LIN {X 0,Y 418.251,Z 298.382,A -85,B 0,C 180,E1 -10100.663,E2 -10100.663} C_VEL
LIN {X 0,Y 418.279,Z 298.377,A -85,B 0,C 180,E1 -10103.782,E2 -10103.782} C_VEL
LIN {X 0,Y 418.312,Z 298.374,A -85,B 0,C 180,E1 -10107.07,E2 -10107.07} C_VEL
LIN {X 0,Y 418.246,Z 298.384,A -85,B 0,C 180,E1 -10110.272,E2 -10110.272} C_VEL
LIN {X 0,Y 418.249,Z 298.383,A -85,B 0,C 180,E1 -10113.677,E2 -10113.677} C_VEL
LIN {X 0,Y 418.241,Z 298.386,A -85,B 0,C 180,E1 -10117.224,E2 -10117.224} C_VEL
LIN {X 0,Y 418.248,Z 298.385,A -85,B 0,C 180,E1 -10119.682,E2 -10119.682} C_VEL
LIN {X 0,Y 418.231,Z 298.386,A -85,B 0,C 180,E1 -10122.321,E2 -10122.321} C_VEL
LIN {X 0,Y 418.237,Z 298.39,A -85,B 0,C 180,E1 -10125.109,E2 -10125.109} C_VEL
LIN {X 0,Y 418.242,Z 298.386,A -85,B 0,C 180,E1 -10127.767,E2 -10127.767} C_VEL
LIN {X 0,Y 418.247,Z 298.385,A -85,B 0,C 180,E1 -10130.62,E2 -10130.62} C_VEL
LIN {X 0,Y 418.245,Z 298.393,A -85,B 0,C 180,E1 -10133.976,E2 -10133.976} C_VEL
LIN {X 0,Y 418.26,Z 298.389,A -85,B 0,C 180,E1 -10137.156,E2 -10137.156} C_VEL
LIN {X 0,Y 418.271,Z 298.384,A -85,B 0,C 180,E1 -10140.895,E2 -10140.895} C_VEL
LIN {X 0,Y 418.335,Z 298.472,A -85,B 0,C 180,E1 -10142.493,E2 -10142.493} C_VEL
LIN {X 0,Y 420.755,Z 310.164,A -85,B 0,C 180,E1 -10144.936,E2 -10144.936} C_VEL
LIN {X 0,Y 421.189,Z 314.876,A -85,B 0,C 180,E1 -10145.87,E2 -10145.87} C_VEL
LIN {X 0,Y 420.116,Z 333.869,A -85,B 0,C 180,E1 -10149.433,E2 -10149.433} C_VEL
LIN {X 0,Y 419.738,Z 340.825,A -85,B 0,C 180,E1 -10150.723,E2 -10150.723} C_VEL
LIN {X 0,Y 423.765,Z 366.097,A -85,B 0,C 180,E1 -10151.423,E2 -10151.423} C_VEL
LIN {X 0,Y 423.972,Z 371.55,A -85,B 0,C 180,E1 -10151.538,E2 -10151.538} C_VEL
LIN {X 0,Y 422.818,Z 450.347,A -85,B 0,C 180,E1 -10152.995,E2 -10152.995} C_VEL
LIN {X 0,Y 422.307,Z 463.22,A -85,B 0,C 180,E1 -10153.41,E2 -10153.41} C_VEL
LIN {X 0,Y 421.668,Z 475.247,A -85,B 0,C 180,E1 -10153.975,E2 -10153.975} C_VEL
LIN {X 0,Y 420.931,Z 487.489,A -85,B 0,C 180,E1 -10154.753,E2 -10154.753} C_VEL
LIN {X 0,Y 420.211,Z 498.894,A -85,B 0,C 180,E1 -10155.697,E2 -10155.697} C_VEL
LIN {X 0,Y 419.4,Z 509.61,A -85,B 0,C 180,E1 -10156.801,E2 -10156.801} C_VEL
LIN {X 0,Y 418.827,Z 518.21,A -85,B 0,C 180,E1 -10157.892,E2 -10157.892} C_VEL
LIN {X 0,Y 418.085,Z 527.537,A -85,B 0,C 180,E1 -10159.344,E2 -10159.344} C_VEL
LIN {X 0,Y 417.632,Z 535.048,A -85,B 0,C 180,E1 -10160.8,E2 -10160.8} C_VEL
LIN {X 0,Y 417.351,Z 541.088,A -85,B 0,C 180,E1 -10162.257,E2 -10162.257} C_VEL
LIN {X 0,Y 417.165,Z 545.849,A -85,B 0,C 180,E1 -10163.708,E2 -10163.708} C_VEL
LIN {X 0,Y 417.107,Z 549.513,A -85,B 0,C 180,E1 -10165.167,E2 -10165.167} C_VEL
LIN {X 0,Y 417.016,Z 551.381,A -85,B 0,C 180,E1 -10166.134,E2 -10166.134} C_VEL
LIN {X 0,Y 417.031,Z 552.79,A -85,B 0,C 180,E1 -10167.101,E2 -10167.101} C_VEL
LIN {X 0,Y 417.069,Z 553.797,A -85,B 0,C 180,E1 -10168.068,E2 -10168.068} C_VEL
LIN {X 0,Y 417.032,Z 554.406,A -85,B 0,C 180,E1 -10169.034,E2 -10169.034} C_VEL
LIN {X 0,Y 417.028,Z 554.587,A -85,B 0,C 180,E1 -10169.999,E2 -10169.999} C_VEL
LIN {X 0,Y 417.032,Z 554.344,A -85,B 0,C 180,E1 -10170.965,E2 -10170.965} C_VEL
LIN {X 0,Y 417.069,Z 553.708,A -85,B 0,C 180,E1 -10171.931,E2 -10171.931} C_VEL
LIN {X 0,Y 417.033,Z 552.671,A -85,B 0,C 180,E1 -10172.897,E2 -10172.897} C_VEL
LIN {X 0,Y 417.016,Z 551.183,A -85,B 0,C 180,E1 -10173.865,E2 -10173.865} C_VEL
LIN {X 0,Y 417.118,Z 548.137,A -85,B 0,C 180,E1 -10175.317,E2 -10175.317} C_VEL
LIN {X 0,Y 417.23,Z 544.008,A -85,B 0,C 180,E1 -10176.771,E2 -10176.771} C_VEL
LIN {X 0,Y 417.491,Z 537.664,A -85,B 0,C 180,E1 -10178.47,E2 -10178.47} C_VEL
LIN {X 0,Y 417.859,Z 530.747,A -85,B 0,C 180,E1 -10179.926,E2 -10179.926} C_VEL
LIN {X 0,Y 418.282,Z 523.68,A -85,B 0,C 180,E1 -10181.14,E2 -10181.14} C_VEL
LIN {X 0,Y 418.918,Z 515.169,A -85,B 0,C 180,E1 -10182.35,E2 -10182.35} C_VEL
LIN {X 0,Y 419.594,Z 504.638,A -85,B 0,C 180,E1 -10183.561,E2 -10183.561} C_VEL
LIN {X 0,Y 420.256,Z 492.783,A -85,B 0,C 180,E1 -10184.651,E2 -10184.651} C_VEL
LIN {X 0,Y 420.974,Z 480.89,A -85,B 0,C 180,E1 -10185.492,E2 -10185.492} C_VEL
LIN {X 0,Y 421.638,Z 468.569,A -85,B 0,C 180,E1 -10186.149,E2 -10186.149} C_VEL
LIN {X 0,Y 422.184,Z 456.025,A -85,B 0,C 180,E1 -10186.625,E2 -10186.625} C_VEL
LIN {X 0,Y 422.534,Z 441.559,A -85,B 0,C 180,E1 -10186.953,E2 -10186.953} C_VEL
LIN {X 0,Y 423.317,Z 366.905,A -85,B 0,C 180,E1 -10188.298,E2 -10188.298} C_VEL
LIN {X 0,Y 419.561,Z 342.148,A -85,B 0,C 180,E1 -10188.937,E2 -10188.937} C_VEL
LIN {X 0,Y 420.631,Z 325.944,A -85,B 0,C 180,E1 -10192.081,E2 -10192.081} C_VEL
LIN {X 0,Y 421.354,Z 314.259,A -85,B 0,C 180,E1 -10194.381,E2 -10194.381} C_VEL
LIN {X 0,Y 419.417,Z 303.717,A -85,B 0,C 180,E1 -10196.63,E2 -10196.63} C_VEL
LIN {X 0,Y 418.333,Z 298.377,A -85,B 0,C 180,E1 -10197.821,E2 -10197.821} C_VEL
LIN {X 0,Y 418.209,Z 298.387,A -85,B 0,C 180,E1 -10201.395,E2 -10201.395} C_VEL
LIN {X 0,Y 418.263,Z 298.383,A -85,B 0,C 180,E1 -10204.58,E2 -10204.58} C_VEL
LIN {X 0,Y 418.223,Z 298.387,A -85,B 0,C 180,E1 -10207.832,E2 -10207.832} C_VEL
LIN {X 0,Y 418.219,Z 298.387,A -85,B 0,C 180,E1 -10210.947,E2 -10210.947} C_VEL
LIN {X 0,Y 418.206,Z 298.387,A -85,B 0,C 180,E1 -10213.729,E2 -10213.729} C_VEL
LIN {X 0,Y 418.212,Z 298.393,A -85,B 0,C 180,E1 -10216.449,E2 -10216.449} C_VEL
LIN {X 0,Y 418.221,Z 298.387,A -85,B 0,C 180,E1 -10219.129,E2 -10219.129} C_VEL
LIN {X 0,Y 418.231,Z 298.385,A -85,B 0,C 180,E1 -10222.165,E2 -10222.165} C_VEL
LIN {X 0,Y 418.261,Z 298.381,A -85,B 0,C 180,E1 -10225.419,E2 -10225.419} C_VEL
LIN {X 0,Y 418.207,Z 298.391,A -85,B 0,C 180,E1 -10228.604,E2 -10228.604} C_VEL
LIN {X 0,Y 418.286,Z 298.377,A -85,B 0,C 180,E1 -10231.936,E2 -10231.936} C_VEL
LIN {X 0,Y 418.284,Z 298.383,A -85,B 0,C 180,E1 -10235.162,E2 -10235.162} C_VEL
LIN {X 0,Y 418.228,Z 298.384,A -85,B 0,C 180,E1 -10238.303,E2 -10238.303} C_VEL
LIN {X 0,Y 418.278,Z 298.383,A -85,B 0,C 180,E1 -10241.383,E2 -10241.383} C_VEL
LIN {X 0,Y 418.297,Z 298.375,A -85,B 0,C 180,E1 -10244.406,E2 -10244.406} C_VEL
LIN {X 0,Y 418.35,Z 298.377,A -85,B 0,C 180,E1 -10247.386,E2 -10247.386} C_VEL
LIN {X 0,Y 418.335,Z 298.371,A -85,B 0,C 180,E1 -10250.329,E2 -10250.329} C_VEL
LIN {X 0,Y 418.507,Z 298.35,A -85,B 0,C 180,E1 -10252.279,E2 -10252.279} C_VEL
LIN {X 0,Y 418.507,Z 298.35,A -85,B 0,C 180,E1 -10254.217,E2 -10254.217} C_VEL
LIN {X 0,Y 418.536,Z 298.348,A -85,B 0,C 180,E1 -10258.076,E2 -10258.076} C_VEL
LIN {X 0,Y 418.664,Z 298.334,A -85,B 0,C 180,E1 -10260,E2 -10260} C_VEL
LIN {X 0,Y 418.496,Z 298.35,A -85,B 0,C 180,E1 -10262.888,E2 -10262.888} C_VEL
LIN {X 0,Y 418.452,Z 298.356,A -85,B 0,C 180,E1 -10266.52,E2 -10266.52} C_VEL
LIN {X 0,Y 418.335,Z 298.374,A -85,B 0,C 180,E1 -10269.672,E2 -10269.672} C_VEL
LIN {X 0,Y 418.341,Z 298.37,A -85,B 0,C 180,E1 -10273.001,E2 -10273.001} C_VEL
LIN {X 0,Y 418.307,Z 298.376,A -85,B 0,C 180,E1 -10276.736,E2 -10276.736} C_VEL
LIN {X 0,Y 418.265,Z 298.382,A -85,B 0,C 180,E1 -10279.791,E2 -10279.791} C_VEL
LIN {X 0,Y 418.227,Z 298.387,A -85,B 0,C 180,E1 -10282.737,E2 -10282.737} C_VEL
LIN {X 0,Y 418.233,Z 298.385,A -85,B 0,C 180,E1 -10285.907,E2 -10285.907} C_VEL
LIN {X 0,Y 418.257,Z 298.381,A -85,B 0,C 180,E1 -10289.163,E2 -10289.163} C_VEL
LIN {X 0,Y 418.254,Z 298.386,A -85,B 0,C 180,E1 -10292.845,E2 -10292.845} C_VEL
LIN {X 0,Y 418.242,Z 298.384,A -85,B 0,C 180,E1 -10296.239,E2 -10296.239} C_VEL
LIN {X 0,Y 418.231,Z 298.384,A -85,B 0,C 180,E1 -10299.685,E2 -10299.685} C_VEL
LIN {X 0,Y 418.221,Z 298.386,A -85,B 0,C 180,E1 -10302.321,E2 -10302.321} C_VEL
LIN {X 0,Y 418.234,Z 298.389,A -85,B 0,C 180,E1 -10305.11,E2 -10305.11} C_VEL
LIN {X 0,Y 418.221,Z 298.385,A -85,B 0,C 180,E1 -10307.766,E2 -10307.766} C_VEL
LIN {X 0,Y 418.239,Z 298.385,A -85,B 0,C 180,E1 -10311.558,E2 -10311.558} C_VEL
LIN {X 0,Y 418.258,Z 298.387,A -85,B 0,C 180,E1 -10315.16,E2 -10315.16} C_VEL
LIN {X 0,Y 418.245,Z 298.387,A -85,B 0,C 180,E1 -10317.473,E2 -10317.473} C_VEL
LIN {X 0,Y 418.262,Z 298.382,A -85,B 0,C 180,E1 -10320.898,E2 -10320.898} C_VEL
LIN {X 0,Y 418.225,Z 298.385,A -85,B 0,C 180,E1 -10324.094,E2 -10324.094} C_VEL
LIN {X 0,Y 418.229,Z 298.388,A -85,B 0,C 180,E1 -10327.264,E2 -10327.264} C_VEL
LIN {X 0,Y 418.285,Z 298.377,A -85,B 0,C 180,E1 -10330.365,E2 -10330.365} C_VEL
LIN {X 0,Y 418.318,Z 298.377,A -85,B 0,C 180,E1 -10333.405,E2 -10333.405} C_VEL
LIN {X 0,Y 418.349,Z 298.369,A -85,B 0,C 180,E1 -10337.001,E2 -10337.001} C_VEL
LIN {X 0,Y 418.323,Z 298.375,A -85,B 0,C 180,E1 -10340.329,E2 -10340.329} C_VEL
LIN {X 0,Y 418.445,Z 298.357,A -85,B 0,C 180,E1 -10343.249,E2 -10343.249} C_VEL
LIN {X 0,Y 418.315,Z 298.373,A -85,B 0,C 180,E1 -10345.182,E2 -10345.182} C_VEL
LIN {X 0,Y 418.533,Z 298.354,A -85,B 0,C 180,E1 -10348.076,E2 -10348.076} C_VEL
LIN {X 0,Y 418.41,Z 298.362,A -85,B 0,C 180,E1 -10350.963,E2 -10350.963} C_VEL
LIN {X 0,Y 418.457,Z 298.356,A -85,B 0,C 180,E1 -10352.889,E2 -10352.889} C_VEL
LIN {X 0,Y 418.473,Z 298.355,A -85,B 0,C 180,E1 -10355.784,E2 -10355.784} C_VEL
LIN {X 0,Y 418.369,Z 298.371,A -85,B 0,C 180,E1 -10358.696,E2 -10358.696} C_VEL
LIN {X 0,Y 418.349,Z 298.376,A -85,B 0,C 180,E1 -10362.615,E2 -10362.615} C_VEL
LIN {X 0,Y 418.305,Z 298.375,A -85,B 0,C 180,E1 -10363.316,E2 -10363.316} C_VEL
LIN {X 0,Y 417.583,Z 298.469,A -85,B 0,C 180,E1 -10364.12,E2 -10364.12} C_VEL
LIN {X 0,Y 414.695,Z 298.824,A -85,B 0,C 180,E1 -10365.425,E2 -10365.425} C_VEL
LIN {X 0,Y 412.29,Z 299.13,A -85,B 0,C 180,E1 -10366.479,E2 -10366.479} C_VEL
LIN {X 0,Y 411.271,Z 299.252,A -85,B 0,C 180,E1 -10367.293,E2 -10367.293} C_VEL
LIN {X 0,Y 411.194,Z 299.26,A -85,B 0,C 180,E1 -10367.569,E2 -10367.569} C_VEL
LIN {X 0,Y 411.192,Z 299.266,A -85,B 0,C 180,E1 -10371.035,E2 -10371.035} C_VEL
LIN {X 0,Y 411.257,Z 299.456,A -85,B 0,C 180,E1 -10374.586,E2 -10374.586} C_VEL
LIN {X 0,Y 413.05,Z 309.513,A -85,B 0,C 180,E1 -10377.075,E2 -10377.075} C_VEL
LIN {X 0,Y 412.957,Z 312.92,A -85,B 0,C 180,E1 -10377.868,E2 -10377.868} C_VEL
LIN {X 0,Y 416.883,Z 333.61,A -85,B 0,C 180,E1 -10378.441,E2 -10378.441} C_VEL
LIN {X 0,Y 415.656,Z 420.17,A -85,B 0,C 180,E1 -10380.043,E2 -10380.043} C_VEL
LIN {X 0,Y 415.177,Z 433.503,A -85,B 0,C 180,E1 -10380.479,E2 -10380.479} C_VEL
LIN {X 0,Y 414.747,Z 446.548,A -85,B 0,C 180,E1 -10381.12,E2 -10381.12} C_VEL
LIN {X 0,Y 414.027,Z 458.605,A -85,B 0,C 180,E1 -10381.924,E2 -10381.924} C_VEL
LIN {X 0,Y 413.292,Z 470.672,A -85,B 0,C 180,E1 -10382.968,E2 -10382.968} C_VEL
LIN {X 0,Y 412.789,Z 480.02,A -85,B 0,C 180,E1 -10383.981,E2 -10383.981} C_VEL
LIN {X 0,Y 412.08,Z 489.365,A -85,B 0,C 180,E1 -10385.218,E2 -10385.218} C_VEL
LIN {X 0,Y 411.368,Z 498.536,A -85,B 0,C 180,E1 -10386.724,E2 -10386.724} C_VEL
LIN {X 0,Y 410.855,Z 506.345,A -85,B 0,C 180,E1 -10388.349,E2 -10388.349} C_VEL
LIN {X 0,Y 410.478,Z 512.736,A -85,B 0,C 180,E1 -10390.066,E2 -10390.066} C_VEL
LIN {X 0,Y 410.236,Z 516.777,A -85,B 0,C 180,E1 -10391.476,E2 -10391.476} C_VEL
LIN {X 0,Y 410.003,Z 520.577,A -85,B 0,C 180,E1 -10393.287,E2 -10393.287} C_VEL
LIN {X 0,Y 409.832,Z 523.05,A -85,B 0,C 180,E1 -10395.324,E2 -10395.324} C_VEL
LIN {X 0,Y 409.822,Z 523.739,A -85,B 0,C 180,E1 -10396.688,E2 -10396.688} C_VEL
LIN {X 0,Y 409.804,Z 523.686,A -85,B 0,C 180,E1 -10398.022,E2 -10398.022} C_VEL
LIN {X 0,Y 409.849,Z 522.874,A -85,B 0,C 180,E1 -10399.336,E2 -10399.336} C_VEL
LIN {X 0,Y 410.076,Z 520.348,A -85,B 0,C 180,E1 -10401.277,E2 -10401.277} C_VEL
LIN {X 0,Y 410.365,Z 516.265,A -85,B 0,C 180,E1 -10403.171,E2 -10403.171} C_VEL
LIN {X 0,Y 410.748,Z 511.185,A -85,B 0,C 180,E1 -10404.845,E2 -10404.845} C_VEL
LIN {X 0,Y 411.254,Z 504.312,A -85,B 0,C 180,E1 -10406.556,E2 -10406.556} C_VEL
LIN {X 0,Y 411.871,Z 496.64,A -85,B 0,C 180,E1 -10408.064,E2 -10408.064} C_VEL
LIN {X 0,Y 412.497,Z 489.141,A -85,B 0,C 180,E1 -10409.26,E2 -10409.26} C_VEL
LIN {X 0,Y 413.144,Z 480.198,A -85,B 0,C 180,E1 -10410.441,E2 -10410.441} C_VEL
LIN {X 0,Y 413.989,Z 469.091,A -85,B 0,C 180,E1 -10411.618,E2 -10411.618} C_VEL
LIN {X 0,Y 414.697,Z 458.601,A -85,B 0,C 180,E1 -10412.51,E2 -10412.51} C_VEL
LIN {X 0,Y 415.357,Z 447.305,A -85,B 0,C 180,E1 -10413.267,E2 -10413.267} C_VEL
LIN {X 0,Y 415.837,Z 434.749,A -85,B 0,C 180,E1 -10413.896,E2 -10413.896} C_VEL
LIN {X 0,Y 416.258,Z 422.566,A -85,B 0,C 180,E1 -10414.314,E2 -10414.314} C_VEL
LIN {X 0,Y 416.73,Z 393.125,A -85,B 0,C 180,E1 -10414.896,E2 -10414.896} C_VEL
LIN {X 0,Y 417.771,Z 332.851,A -85,B 0,C 180,E1 -10416.022,E2 -10416.022} C_VEL
LIN {X 0,Y 413.467,Z 312.572,A -85,B 0,C 180,E1 -10416.669,E2 -10416.669} C_VEL
LIN {X 0,Y 413.236,Z 308.374,A -85,B 0,C 180,E1 -10417.501,E2 -10417.501} C_VEL
LIN {X 0,Y 411.241,Z 299.26,A -85,B 0,C 180,E1 -10419.426,E2 -10419.426} C_VEL
LIN {X 0,Y 411.266,Z 299.262,A -85,B 0,C 180,E1 -10423.131,E2 -10423.131} C_VEL
LIN {X 0,Y 411.308,Z 299.252,A -85,B 0,C 180,E1 -10426.896,E2 -10426.896} C_VEL
LIN {X 0,Y 411.294,Z 299.253,A -85,B 0,C 180,E1 -10430.161,E2 -10430.161} C_VEL
LIN {X 0,Y 411.485,Z 299.23,A -85,B 0,C 180,E1 -10432.146,E2 -10432.146} C_VEL
LIN {X 0,Y 411.473,Z 299.232,A -85,B 0,C 180,E1 -10434.118,E2 -10434.118} C_VEL
LIN {X 0,Y 411.513,Z 299.224,A -85,B 0,C 180,E1 -10438.042,E2 -10438.042} C_VEL
LIN {X 0,Y 411.642,Z 299.21,A -85,B 0,C 180,E1 -10440,E2 -10440} C_VEL
LIN {X 0,Y 411.459,Z 299.229,A -85,B 0,C 180,E1 -10442.937,E2 -10442.937} C_VEL
LIN {X 0,Y 411.46,Z 299.234,A -85,B 0,C 180,E1 -10445.882,E2 -10445.882} C_VEL
LIN {X 0,Y 411.353,Z 299.242,A -85,B 0,C 180,E1 -10448.845,E2 -10448.845} C_VEL
LIN {X 0,Y 411.285,Z 299.252,A -85,B 0,C 180,E1 -10451.833,E2 -10451.833} C_VEL
LIN {X 0,Y 411.263,Z 299.256,A -85,B 0,C 180,E1 -10454.852,E2 -10454.852} C_VEL
LIN {X 0,Y 411.247,Z 299.252,A -85,B 0,C 180,E1 -10457.915,E2 -10457.915} C_VEL
LIN {X 0,Y 411.198,Z 299.26,A -85,B 0,C 180,E1 -10461.034,E2 -10461.034} C_VEL
LIN {X 0,Y 411.222,Z 299.258,A -85,B 0,C 180,E1 -10464.216,E2 -10464.216} C_VEL
LIN {X 0,Y 411.261,Z 299.249,A -85,B 0,C 180,E1 -10467.477,E2 -10467.477} C_VEL
LIN {X 0,Y 411.191,Z 299.264,A -85,B 0,C 180,E1 -10470.847,E2 -10470.847} C_VEL
LIN {X 0,Y 411.206,Z 299.26,A -85,B 0,C 180,E1 -10474.333,E2 -10474.333} C_VEL
LIN {X 0,Y 411.195,Z 299.26,A -85,B 0,C 180,E1 -10477.974,E2 -10477.974} C_VEL
LIN {X 0,Y 411.165,Z 299.268,A -85,B 0,C 180,E1 -10481.228,E2 -10481.228} C_VEL
LIN {X 0,Y 411.178,Z 299.265,A -85,B 0,C 180,E1 -10484.49,E2 -10484.49} C_VEL
LIN {X 0,Y 411.179,Z 299.264,A -85,B 0,C 180,E1 -10488.194,E2 -10488.194} C_VEL
LIN {X 0,Y 411.213,Z 299.261,A -85,B 0,C 180,E1 -10490.775,E2 -10490.775} C_VEL
LIN {X 0,Y 411.2,Z 299.267,A -85,B 0,C 180,E1 -10494.471,E2 -10494.471} C_VEL
LIN {X 0,Y 411.209,Z 299.267,A -85,B 0,C 180,E1 -10496.873,E2 -10496.873} C_VEL
LIN {X 0,Y 411.235,Z 299.261,A -85,B 0,C 180,E1 -10500.644,E2 -10500.644} C_VEL
LIN {X 0,Y 411.296,Z 299.362,A -85,B 0,C 180,E1 -10502.179,E2 -10502.179} C_VEL
LIN {X 0,Y 413.562,Z 310.096,A -85,B 0,C 180,E1 -10504.478,E2 -10504.478} C_VEL
LIN {X 0,Y 414.314,Z 314.766,A -85,B 0,C 180,E1 -10505.443,E2 -10505.443} C_VEL
LIN {X 0,Y 413.476,Z 329.694,A -85,B 0,C 180,E1 -10508.303,E2 -10508.303} C_VEL
LIN {X 0,Y 412.854,Z 340.517,A -85,B 0,C 180,E1 -10510.354,E2 -10510.354} C_VEL
LIN {X 0,Y 416.827,Z 364.726,A -85,B 0,C 180,E1 -10511.046,E2 -10511.046} C_VEL
LIN {X 0,Y 417.328,Z 371.186,A -85,B 0,C 180,E1 -10511.199,E2 -10511.199} C_VEL
LIN {X 0,Y 416.084,Z 449.753,A -85,B 0,C 180,E1 -10512.68,E2 -10512.68} C_VEL
LIN {X 0,Y 415.553,Z 462.683,A -85,B 0,C 180,E1 -10513.101,E2 -10513.101} C_VEL
LIN {X 0,Y 414.857,Z 475.303,A -85,B 0,C 180,E1 -10513.705,E2 -10513.705} C_VEL
LIN {X 0,Y 414.065,Z 487.431,A -85,B 0,C 180,E1 -10514.494,E2 -10514.494} C_VEL
LIN {X 0,Y 413.274,Z 499.279,A -85,B 0,C 180,E1 -10515.498,E2 -10515.498} C_VEL
LIN {X 0,Y 412.482,Z 509.488,A -85,B 0,C 180,E1 -10516.576,E2 -10516.576} C_VEL
LIN {X 0,Y 411.872,Z 518.065,A -85,B 0,C 180,E1 -10517.684,E2 -10517.684} C_VEL
LIN {X 0,Y 411.078,Z 527.364,A -85,B 0,C 180,E1 -10519.16,E2 -10519.16} C_VEL
LIN {X 0,Y 410.595,Z 534.864,A -85,B 0,C 180,E1 -10520.641,E2 -10520.641} C_VEL
LIN {X 0,Y 410.288,Z 540.892,A -85,B 0,C 180,E1 -10522.123,E2 -10522.123} C_VEL
LIN {X 0,Y 410.058,Z 546.081,A -85,B 0,C 180,E1 -10523.755,E2 -10523.755} C_VEL
LIN {X 0,Y 410.018,Z 549.288,A -85,B 0,C 180,E1 -10525.083,E2 -10525.083} C_VEL
LIN {X 0,Y 409.933,Z 551.142,A -85,B 0,C 180,E1 -10526.067,E2 -10526.067} C_VEL
LIN {X 0,Y 409.996,Z 553.547,A -85,B 0,C 180,E1 -10528.035,E2 -10528.035} C_VEL
LIN {X 0,Y 409.955,Z 554.15,A -85,B 0,C 180,E1 -10529.017,E2 -10529.017} C_VEL
LIN {X 0,Y 409.949,Z 554.318,A -85,B 0,C 180,E1 -10529.999,E2 -10529.999} C_VEL
LIN {X 0,Y 409.955,Z 554.07,A -85,B 0,C 180,E1 -10530.982,E2 -10530.982} C_VEL
LIN {X 0,Y 409.996,Z 553.427,A -85,B 0,C 180,E1 -10531.964,E2 -10531.964} C_VEL
LIN {X 0,Y 409.932,Z 552.382,A -85,B 0,C 180,E1 -10532.948,E2 -10532.948} C_VEL
LIN {X 0,Y 409.935,Z 550.88,A -85,B 0,C 180,E1 -10533.932,E2 -10533.932} C_VEL
LIN {X 0,Y 410.013,Z 547.813,A -85,B 0,C 180,E1 -10535.409,E2 -10535.409} C_VEL
LIN {X 0,Y 410.162,Z 543.664,A -85,B 0,C 180,E1 -10536.888,E2 -10536.888} C_VEL
LIN {X 0,Y 410.423,Z 537.292,A -85,B 0,C 180,E1 -10538.617,E2 -10538.617} C_VEL
LIN {X 0,Y 410.829,Z 530.345,A -85,B 0,C 180,E1 -10540.098,E2 -10540.098} C_VEL
LIN {X 0,Y 411.289,Z 523.242,A -85,B 0,C 180,E1 -10541.332,E2 -10541.332} C_VEL
LIN {X 0,Y 411.926,Z 514.673,A -85,B 0,C 180,E1 -10542.563,E2 -10542.563} C_VEL
LIN {X 0,Y 412.632,Z 504.07,A -85,B 0,C 180,E1 -10543.794,E2 -10543.794} C_VEL
LIN {X 0,Y 413.363,Z 492.127,A -85,B 0,C 180,E1 -10544.901,E2 -10544.901} C_VEL
LIN {X 0,Y 414.083,Z 480.083,A -85,B 0,C 180,E1 -10545.756,E2 -10545.756} C_VEL
LIN {X 0,Y 414.838,Z 467.602,A -85,B 0,C 180,E1 -10546.421,E2 -10546.421} C_VEL
LIN {X 0,Y 415.33,Z 454.641,A -85,B 0,C 180,E1 -10546.907,E2 -10546.907} C_VEL
LIN {X 0,Y 415.712,Z 437.732,A -85,B 0,C 180,E1 -10547.271,E2 -10547.271} C_VEL
LIN {X 0,Y 416.53,Z 367.926,A -85,B 0,C 180,E1 -10548.553,E2 -10548.553} C_VEL
LIN {X 0,Y 412.622,Z 341.914,A -85,B 0,C 180,E1 -10549.236,E2 -10549.236} C_VEL
LIN {X 0,Y 413.811,Z 324.271,A -85,B 0,C 180,E1 -10552.728,E2 -10552.728} C_VEL
LIN {X 0,Y 414.367,Z 315.186,A -85,B 0,C 180,E1 -10554.553,E2 -10554.553} C_VEL
LIN {X 0,Y 412.374,Z 304.623,A -85,B 0,C 180,E1 -10556.848,E2 -10556.848} C_VEL
LIN {X 0,Y 411.271,Z 299.258,A -85,B 0,C 180,E1 -10558.098,E2 -10558.098} C_VEL
LIN {X 0,Y 411.18,Z 299.262,A -85,B 0,C 180,E1 -10561.283,E2 -10561.283} C_VEL
LIN {X 0,Y 411.204,Z 299.265,A -85,B 0,C 180,E1 -10564.333,E2 -10564.333} C_VEL
LIN {X 0,Y 411.189,Z 299.264,A -85,B 0,C 180,E1 -10567.973,E2 -10567.973} C_VEL
LIN {X 0,Y 411.16,Z 299.265,A -85,B 0,C 180,E1 -10571.228,E2 -10571.228} C_VEL
LIN {X 0,Y 411.173,Z 299.271,A -85,B 0,C 180,E1 -10574.49,E2 -10574.49} C_VEL
LIN {X 0,Y 411.175,Z 299.266,A -85,B 0,C 180,E1 -10578.194,E2 -10578.194} C_VEL
LIN {X 0,Y 411.22,Z 299.263,A -85,B 0,C 180,E1 -10580.776,E2 -10580.776} C_VEL
LIN {X 0,Y 411.195,Z 299.264,A -85,B 0,C 180,E1 -10584.471,E2 -10584.471} C_VEL
LIN {X 0,Y 411.202,Z 299.266,A -85,B 0,C 180,E1 -10586.873,E2 -10586.873} C_VEL
LIN {X 0,Y 411.227,Z 299.26,A -85,B 0,C 180,E1 -10590.644,E2 -10590.644} C_VEL
LIN {X 0,Y 411.232,Z 299.257,A -85,B 0,C 180,E1 -10593.619,E2 -10593.619} C_VEL
LIN {X 0,Y 411.198,Z 299.264,A -85,B 0,C 180,E1 -10596.852,E2 -10596.852} C_VEL
LIN {X 0,Y 411.209,Z 299.258,A -85,B 0,C 180,E1 -10600.05,E2 -10600.05} C_VEL
LIN {X 0,Y 411.257,Z 299.258,A -85,B 0,C 180,E1 -10603.131,E2 -10603.131} C_VEL
LIN {X 0,Y 411.299,Z 299.249,A -85,B 0,C 180,E1 -10606.896,E2 -10606.896} C_VEL
LIN {X 0,Y 411.287,Z 299.249,A -85,B 0,C 180,E1 -10610.161,E2 -10610.161} C_VEL
LIN {X 0,Y 411.454,Z 299.231,A -85,B 0,C 180,E1 -10613.133,E2 -10613.133} C_VEL
LIN {X 0,Y 411.304,Z 299.249,A -85,B 0,C 180,E1 -10615.099,E2 -10615.099} C_VEL
LIN {X 0,Y 411.505,Z 299.225,A -85,B 0,C 180,E1 -10618.043,E2 -10618.043} C_VEL
LIN {X 0,Y 411.634,Z 299.21,A -85,B 0,C 180,E1 -10620,E2 -10620} C_VEL
LIN {X 0,Y 411.453,Z 299.228,A -85,B 0,C 180,E1 -10622.938,E2 -10622.938} C_VEL
LIN {X 0,Y 411.416,Z 299.234,A -85,B 0,C 180,E1 -10626.518,E2 -10626.518} C_VEL
LIN {X 0,Y 411.287,Z 299.254,A -85,B 0,C 180,E1 -10629.839,E2 -10629.839} C_VEL
LIN {X 0,Y 411.3,Z 299.247,A -85,B 0,C 180,E1 -10633.105,E2 -10633.105} C_VEL
LIN {X 0,Y 411.252,Z 299.254,A -85,B 0,C 180,E1 -10636.889,E2 -10636.889} C_VEL
LIN {X 0,Y 411.226,Z 299.26,A -85,B 0,C 180,E1 -10639.987,E2 -10639.987} C_VEL
LIN {X 0,Y 411.191,Z 299.261,A -85,B 0,C 180,E1 -10643.149,E2 -10643.149} C_VEL
LIN {X 0,Y 411.191,Z 299.268,A -85,B 0,C 180,E1 -10646.385,E2 -10646.385} C_VEL
LIN {X 0,Y 411.194,Z 299.26,A -85,B 0,C 180,E1 -10649.714,E2 -10649.714} C_VEL
LIN {X 0,Y 411.203,Z 299.261,A -85,B 0,C 180,E1 -10653.157,E2 -10653.157} C_VEL
LIN {X 0,Y 411.189,Z 299.266,A -85,B 0,C 180,E1 -10656.553,E2 -10656.553} C_VEL
LIN {X 0,Y 411.196,Z 299.26,A -85,B 0,C 180,E1 -10659.726,E2 -10659.726} C_VEL
LIN {X 0,Y 411.168,Z 299.268,A -85,B 0,C 180,E1 -10663.135,E2 -10663.135} C_VEL
LIN {X 0,Y 411.163,Z 299.264,A -85,B 0,C 180,E1 -10665.882,E2 -10665.882} C_VEL
LIN {X 0,Y 411.149,Z 299.27,A -85,B 0,C 180,E1 -10668.775,E2 -10668.775} C_VEL
LIN {X 0,Y 411.187,Z 299.261,A -85,B 0,C 180,E1 -10672.026,E2 -10672.026} C_VEL
LIN {X 0,Y 411.204,Z 299.261,A -85,B 0,C 180,E1 -10675.667,E2 -10675.667} C_VEL
LIN {X 0,Y 411.189,Z 299.266,A -85,B 0,C 180,E1 -10679.153,E2 -10679.153} C_VEL
LIN {X 0,Y 411.177,Z 299.27,A -85,B 0,C 180,E1 -10681.408,E2 -10681.408} C_VEL
LIN {X 0,Y 411.189,Z 299.262,A -85,B 0,C 180,E1 -10684.942,E2 -10684.942} C_VEL
LIN {X 0,Y 411.205,Z 299.262,A -85,B 0,C 180,E1 -10687.914,E2 -10687.914} C_VEL
LIN {X 0,Y 411.22,Z 299.258,A -85,B 0,C 180,E1 -10691.052,E2 -10691.052} C_VEL
LIN {X 0,Y 411.254,Z 299.256,A -85,B 0,C 180,E1 -10694.132,E2 -10694.132} C_VEL
LIN {X 0,Y 411.306,Z 299.247,A -85,B 0,C 180,E1 -10697.166,E2 -10697.166} C_VEL
LIN {X 0,Y 411.278,Z 299.254,A -85,B 0,C 180,E1 -10700.162,E2 -10700.162} C_VEL
LIN {X 0,Y 411.394,Z 299.235,A -85,B 0,C 180,E1 -10703.133,E2 -10703.133} C_VEL
LIN {X 0,Y 411.287,Z 299.249,A -85,B 0,C 180,E1 -10705.099,E2 -10705.099} C_VEL
LIN {X 0,Y 411.501,Z 299.229,A -85,B 0,C 180,E1 -10708.043,E2 -10708.043} C_VEL
LIN {X 0,Y 411.38,Z 299.237,A -85,B 0,C 180,E1 -10710.979,E2 -10710.979} C_VEL
LIN {X 0,Y 411.416,Z 299.233,A -85,B 0,C 180,E1 -10712.938,E2 -10712.938} C_VEL
LIN {X 0,Y 411.42,Z 299.234,A -85,B 0,C 180,E1 -10715.883,E2 -10715.883} C_VEL
LIN {X 0,Y 411.308,Z 299.249,A -85,B 0,C 180,E1 -10718.847,E2 -10718.847} C_VEL
LIN {X 0,Y 411.269,Z 299.252,A -85,B 0,C 180,E1 -10721.834,E2 -10721.834} C_VEL
LIN {X 0,Y 411.212,Z 299.262,A -85,B 0,C 180,E1 -10724.855,E2 -10724.855} C_VEL
LIN {X 0,Y 411.194,Z 299.26,A -85,B 0,C 180,E1 -10727.569,E2 -10727.569} C_VEL
LIN {X 0,Y 410.536,Z 299.349,A -85,B 0,C 180,E1 -10728.387,E2 -10728.387} C_VEL
LIN {X 0,Y 407.665,Z 299.701,A -85,B 0,C 180,E1 -10729.717,E2 -10729.717} C_VEL
LIN {X 0,Y 405.237,Z 300.01,A -85,B 0,C 180,E1 -10730.79,E2 -10730.79} C_VEL
LIN {X 0,Y 404.208,Z 300.134,A -85,B 0,C 180,E1 -10731.62,E2 -10731.62} C_VEL
LIN {X 0,Y 404.132,Z 300.143,A -85,B 0,C 180,E1 -10731.902,E2 -10731.902} C_VEL
LIN {X 0,Y 404.185,Z 300.154,A -85,B 0,C 180,E1 -10734.323,E2 -10734.323} C_VEL
LIN {X 0,Y 406.106,Z 310.893,A -85,B 0,C 180,E1 -10737.019,E2 -10737.019} C_VEL
LIN {X 0,Y 406.035,Z 313.122,A -85,B 0,C 180,E1 -10737.547,E2 -10737.547} C_VEL
LIN {X 0,Y 410.073,Z 333.956,A -85,B 0,C 180,E1 -10738.153,E2 -10738.153} C_VEL
LIN {X 0,Y 408.782,Z 420.734,A -85,B 0,C 180,E1 -10739.793,E2 -10739.793} C_VEL
LIN {X 0,Y 408.287,Z 434.353,A -85,B 0,C 180,E1 -10740.253,E2 -10740.253} C_VEL
LIN {X 0,Y 407.857,Z 446.922,A -85,B 0,C 180,E1 -10740.888,E2 -10740.888} C_VEL
LIN {X 0,Y 407.128,Z 458.844,A -85,B 0,C 180,E1 -10741.697,E2 -10741.697} C_VEL
LIN {X 0,Y 406.387,Z 470.461,A -85,B 0,C 180,E1 -10742.714,E2 -10742.714} C_VEL
LIN {X 0,Y 405.826,Z 480.131,A -85,B 0,C 180,E1 -10743.771,E2 -10743.771} C_VEL
LIN {X 0,Y 405.053,Z 490.167,A -85,B 0,C 180,E1 -10745.13,E2 -10745.13} C_VEL
LIN {X 0,Y 404.384,Z 498.631,A -85,B 0,C 180,E1 -10746.548,E2 -10746.548} C_VEL
LIN {X 0,Y 403.854,Z 505.525,A -85,B 0,C 180,E1 -10747.972,E2 -10747.972} C_VEL
LIN {X 0,Y 403.484,Z 511.051,A -85,B 0,C 180,E1 -10749.387,E2 -10749.387} C_VEL
LIN {X 0,Y 403.261,Z 515.424,A -85,B 0,C 180,E1 -10750.789,E2 -10750.789} C_VEL
LIN {X 0,Y 403.049,Z 518.784,A -85,B 0,C 180,E1 -10752.17,E2 -10752.17} C_VEL
LIN {X 0,Y 402.861,Z 521.298,A -85,B 0,C 180,E1 -10753.557,E2 -10753.557} C_VEL
LIN {X 0,Y 402.781,Z 522.333,A -85,B 0,C 180,E1 -10754.324,E2 -10754.324} C_VEL
LIN {X 0,Y 402.72,Z 523.611,A -85,B 0,C 180,E1 -10755.728,E2 -10755.728} C_VEL
LIN {X 0,Y 402.732,Z 524.084,A -85,B 0,C 180,E1 -10757.133,E2 -10757.133} C_VEL
LIN {X 0,Y 402.736,Z 523.697,A -85,B 0,C 180,E1 -10758.624,E2 -10758.624} C_VEL
LIN {X 0,Y 402.812,Z 522.38,A -85,B 0,C 180,E1 -10760.147,E2 -10760.147} C_VEL
LIN {X 0,Y 403.051,Z 520.062,A -85,B 0,C 180,E1 -10761.69,E2 -10761.69} C_VEL
LIN {X 0,Y 403.32,Z 516.588,A -85,B 0,C 180,E1 -10763.28,E2 -10763.28} C_VEL
LIN {X 0,Y 403.714,Z 511.689,A -85,B 0,C 180,E1 -10764.937,E2 -10764.937} C_VEL
LIN {X 0,Y 404.215,Z 505.346,A -85,B 0,C 180,E1 -10766.571,E2 -10766.571} C_VEL
LIN {X 0,Y 404.845,Z 497.769,A -85,B 0,C 180,E1 -10768.12,E2 -10768.12} C_VEL
LIN {X 0,Y 405.638,Z 489.052,A -85,B 0,C 180,E1 -10769.55,E2 -10769.55} C_VEL
LIN {X 0,Y 406.441,Z 478.743,A -85,B 0,C 180,E1 -10770.9,E2 -10770.9} C_VEL
LIN {X 0,Y 407.271,Z 467.815,A -85,B 0,C 180,E1 -10772.047,E2 -10772.047} C_VEL
LIN {X 0,Y 408.007,Z 456.54,A -85,B 0,C 180,E1 -10772.979,E2 -10772.979} C_VEL
LIN {X 0,Y 408.822,Z 443.574,A -85,B 0,C 180,E1 -10773.794,E2 -10773.794} C_VEL
LIN {X 0,Y 409.275,Z 430.993,A -85,B 0,C 180,E1 -10774.372,E2 -10774.372} C_VEL
LIN {X 0,Y 409.629,Z 417.525,A -85,B 0,C 180,E1 -10774.767,E2 -10774.767} C_VEL
LIN {X 0,Y 411.117,Z 333.656,A -85,B 0,C 180,E1 -10776.367,E2 -10776.367} C_VEL
LIN {X 0,Y 406.696,Z 312.873,A -85,B 0,C 180,E1 -10777.052,E2 -10777.052} C_VEL
LIN {X 0,Y 405.897,Z 307.647,A -85,B 0,C 180,E1 -10778.144,E2 -10778.144} C_VEL
LIN {X 0,Y 404.208,Z 300.137,A -85,B 0,C 180,E1 -10779.808,E2 -10779.808} C_VEL
LIN {X 0,Y 404.219,Z 300.14,A -85,B 0,C 180,E1 -10782.993,E2 -10782.993} C_VEL
LIN {X 0,Y 404.285,Z 300.127,A -85,B 0,C 180,E1 -10786.939,E2 -10786.939} C_VEL
LIN {X 0,Y 404.259,Z 300.13,A -85,B 0,C 180,E1 -10789.988,E2 -10789.988} C_VEL
LIN {X 0,Y 404.412,Z 300.109,A -85,B 0,C 180,E1 -10793.012,E2 -10793.012} C_VEL
LIN {X 0,Y 404.282,Z 300.125,A -85,B 0,C 180,E1 -10795.013,E2 -10795.013} C_VEL
LIN {X 0,Y 404.482,Z 300.1,A -85,B 0,C 180,E1 -10798.008,E2 -10798.008} C_VEL
LIN {X 0,Y 404.611,Z 300.086,A -85,B 0,C 180,E1 -10800,E2 -10800} C_VEL
LIN {X 0,Y 404.417,Z 300.106,A -85,B 0,C 180,E1 -10802.988,E2 -10802.988} C_VEL
LIN {X 0,Y 404.407,Z 300.111,A -85,B 0,C 180,E1 -10805.985,E2 -10805.985} C_VEL
LIN {X 0,Y 404.29,Z 300.121,A -85,B 0,C 180,E1 -10809.001,E2 -10809.001} C_VEL
LIN {X 0,Y 404.257,Z 300.129,A -85,B 0,C 180,E1 -10812.041,E2 -10812.041} C_VEL
LIN {X 0,Y 404.208,Z 300.133,A -85,B 0,C 180,E1 -10815.118,E2 -10815.118} C_VEL
LIN {X 0,Y 404.206,Z 300.132,A -85,B 0,C 180,E1 -10818.238,E2 -10818.238} C_VEL
LIN {X 0,Y 404.14,Z 300.138,A -85,B 0,C 180,E1 -10821.419,E2 -10821.419} C_VEL
LIN {X 0,Y 404.176,Z 300.135,A -85,B 0,C 180,E1 -10824.666,E2 -10824.666} C_VEL
LIN {X 0,Y 404.197,Z 300.128,A -85,B 0,C 180,E1 -10827.999,E2 -10827.999} C_VEL
LIN {X 0,Y 404.14,Z 300.139,A -85,B 0,C 180,E1 -10831.558,E2 -10831.558} C_VEL
LIN {X 0,Y 404.185,Z 300.136,A -85,B 0,C 180,E1 -10835.016,E2 -10835.016} C_VEL
LIN {X 0,Y 404.154,Z 300.139,A -85,B 0,C 180,E1 -10838.757,E2 -10838.757} C_VEL
LIN {X 0,Y 404.125,Z 300.148,A -85,B 0,C 180,E1 -10841.6,E2 -10841.6} C_VEL
LIN {X 0,Y 404.147,Z 300.141,A -85,B 0,C 180,E1 -10844.522,E2 -10844.522} C_VEL
LIN {X 0,Y 404.138,Z 300.147,A -85,B 0,C 180,E1 -10847.295,E2 -10847.295} C_VEL
LIN {X 0,Y 404.171,Z 300.14,A -85,B 0,C 180,E1 -10849.955,E2 -10849.955} C_VEL
LIN {X 0,Y 404.138,Z 300.147,A -85,B 0,C 180,E1 -10853.125,E2 -10853.125} C_VEL
LIN {X 0,Y 404.147,Z 300.148,A -85,B 0,C 180,E1 -10856.188,E2 -10856.188} C_VEL
LIN {X 0,Y 404.148,Z 300.144,A -85,B 0,C 180,E1 -10859.715,E2 -10859.715} C_VEL
LIN {X 0,Y 404.248,Z 300.329,A -85,B 0,C 180,E1 -10861.863,E2 -10861.863} C_VEL
LIN {X 0,Y 406.727,Z 311.916,A -85,B 0,C 180,E1 -10864.406,E2 -10864.406} C_VEL
LIN {X 0,Y 407.434,Z 317.374,A -85,B 0,C 180,E1 -10865.544,E2 -10865.544} C_VEL
LIN {X 0,Y 406.225,Z 336.543,A -85,B 0,C 180,E1 -10869.258,E2 -10869.258} C_VEL
LIN {X 0,Y 405.995,Z 340.179,A -85,B 0,C 180,E1 -10869.957,E2 -10869.957} C_VEL
LIN {X 0,Y 409.814,Z 363.004,A -85,B 0,C 180,E1 -10870.644,E2 -10870.644} C_VEL
LIN {X 0,Y 410.681,Z 371.616,A -85,B 0,C 180,E1 -10870.863,E2 -10870.863} C_VEL
LIN {X 0,Y 409.328,Z 450.459,A -85,B 0,C 180,E1 -10872.385,E2 -10872.385} C_VEL
LIN {X 0,Y 408.769,Z 463.806,A -85,B 0,C 180,E1 -10872.844,E2 -10872.844} C_VEL
LIN {X 0,Y 408.066,Z 475.506,A -85,B 0,C 180,E1 -10873.426,E2 -10873.426} C_VEL
LIN {X 0,Y 407.224,Z 487.48,A -85,B 0,C 180,E1 -10874.227,E2 -10874.227} C_VEL
LIN {X 0,Y 406.386,Z 499.245,A -85,B 0,C 180,E1 -10875.247,E2 -10875.247} C_VEL
LIN {X 0,Y 405.464,Z 510.445,A -85,B 0,C 180,E1 -10876.471,E2 -10876.471} C_VEL
LIN {X 0,Y 404.762,Z 519.59,A -85,B 0,C 180,E1 -10877.719,E2 -10877.719} C_VEL
LIN {X 0,Y 403.972,Z 528.574,A -85,B 0,C 180,E1 -10879.221,E2 -10879.221} C_VEL
LIN {X 0,Y 403.481,Z 535.794,A -85,B 0,C 180,E1 -10880.728,E2 -10880.728} C_VEL
LIN {X 0,Y 403.227,Z 540.695,A -85,B 0,C 180,E1 -10881.984,E2 -10881.984} C_VEL
LIN {X 0,Y 402.979,Z 546.174,A -85,B 0,C 180,E1 -10883.767,E2 -10883.767} C_VEL
LIN {X 0,Y 402.931,Z 549.068,A -85,B 0,C 180,E1 -10884.996,E2 -10884.996} C_VEL
LIN {X 0,Y 402.854,Z 550.907,A -85,B 0,C 180,E1 -10885.998,E2 -10885.998} C_VEL
LIN {X 0,Y 402.906,Z 553.299,A -85,B 0,C 180,E1 -10888,E2 -10888} C_VEL
LIN {X 0,Y 402.882,Z 553.895,A -85,B 0,C 180,E1 -10889,E2 -10889} C_VEL
LIN {X 0,Y 402.872,Z 554.048,A -85,B 0,C 180,E1 -10889.999,E2 -10889.999} C_VEL
LIN {X 0,Y 402.881,Z 553.791,A -85,B 0,C 180,E1 -10890.999,E2 -10890.999} C_VEL
LIN {X 0,Y 402.907,Z 553.139,A -85,B 0,C 180,E1 -10891.999,E2 -10891.999} C_VEL
LIN {X 0,Y 402.833,Z 552.081,A -85,B 0,C 180,E1 -10893,E2 -10893} C_VEL
LIN {X 0,Y 402.856,Z 550.561,A -85,B 0,C 180,E1 -10894.001,E2 -10894.001} C_VEL
LIN {X 0,Y 402.91,Z 547.47,A -85,B 0,C 180,E1 -10895.505,E2 -10895.505} C_VEL
LIN {X 0,Y 403.074,Z 543.296,A -85,B 0,C 180,E1 -10897.01,E2 -10897.01} C_VEL
LIN {X 0,Y 403.372,Z 536.895,A -85,B 0,C 180,E1 -10898.768,E2 -10898.768} C_VEL
LIN {X 0,Y 403.775,Z 529.912,A -85,B 0,C 180,E1 -10900.276,E2 -10900.276} C_VEL
LIN {X 0,Y 404.407,Z 521.152,A -85,B 0,C 180,E1 -10901.782,E2 -10901.782} C_VEL
LIN {X 0,Y 405.042,Z 512.163,A -85,B 0,C 180,E1 -10903.036,E2 -10903.036} C_VEL
LIN {X 0,Y 405.894,Z 501.076,A -85,B 0,C 180,E1 -10904.284,E2 -10904.284} C_VEL
LIN {X 0,Y 406.574,Z 489.838,A -85,B 0,C 180,E1 -10905.284,E2 -10905.284} C_VEL
LIN {X 0,Y 407.351,Z 477.27,A -85,B 0,C 180,E1 -10906.152,E2 -10906.152} C_VEL
LIN {X 0,Y 408.053,Z 464.438,A -85,B 0,C 180,E1 -10906.799,E2 -10906.799} C_VEL
LIN {X 0,Y 408.617,Z 450.916,A -85,B 0,C 180,E1 -10907.258,E2 -10907.258} C_VEL
LIN {X 0,Y 409.681,Z 368.378,A -85,B 0,C 180,E1 -10908.829,E2 -10908.829} C_VEL
LIN {X 0,Y 405.705,Z 341.694,A -85,B 0,C 180,E1 -10909.544,E2 -10909.544} C_VEL
LIN {X 0,Y 406.845,Z 325.179,A -85,B 0,C 180,E1 -10912.871,E2 -10912.871} C_VEL
LIN {X 0,Y 407.377,Z 316.083,A -85,B 0,C 180,E1 -10914.73,E2 -10914.73} C_VEL
LIN {X 0,Y 405.155,Z 304.526,A -85,B 0,C 180,E1 -10917.297,E2 -10917.297} C_VEL
LIN {X 0,Y 404.218,Z 300.135,A -85,B 0,C 180,E1 -10918.35,E2 -10918.35} C_VEL
LIN {X 0,Y 404.137,Z 300.141,A -85,B 0,C 180,E1 -10921.557,E2 -10921.557} C_VEL
LIN {X 0,Y 404.182,Z 300.134,A -85,B 0,C 180,E1 -10925.015,E2 -10925.015} C_VEL
LIN {X 0,Y 404.147,Z 300.141,A -85,B 0,C 180,E1 -10928.757,E2 -10928.757} C_VEL
LIN {X 0,Y 404.119,Z 300.142,A -85,B 0,C 180,E1 -10931.599,E2 -10931.599} C_VEL
LIN {X 0,Y 404.143,Z 300.146,A -85,B 0,C 180,E1 -10934.522,E2 -10934.522} C_VEL
LIN {X 0,Y 404.136,Z 300.14,A -85,B 0,C 180,E1 -10937.295,E2 -10937.295} C_VEL
LIN {X 0,Y 404.164,Z 300.137,A -85,B 0,C 180,E1 -10939.955,E2 -10939.955} C_VEL
LIN {X 0,Y 404.135,Z 300.142,A -85,B 0,C 180,E1 -10943.124,E2 -10943.124} C_VEL
LIN {X 0,Y 404.14,Z 300.14,A -85,B 0,C 180,E1 -10946.187,E2 -10946.187} C_VEL
LIN {X 0,Y 404.14,Z 300.139,A -85,B 0,C 180,E1 -10949.715,E2 -10949.715} C_VEL
LIN {X 0,Y 404.19,Z 300.139,A -85,B 0,C 180,E1 -10953.123,E2 -10953.123} C_VEL
LIN {X 0,Y 404.172,Z 300.139,A -85,B 0,C 180,E1 -10955.334,E2 -10955.334} C_VEL
LIN {X 0,Y 404.133,Z 300.141,A -85,B 0,C 180,E1 -10958.58,E2 -10958.58} C_VEL
LIN {X 0,Y 404.205,Z 300.133,A -85,B 0,C 180,E1 -10961.762,E2 -10961.762} C_VEL
LIN {X 0,Y 404.201,Z 300.134,A -85,B 0,C 180,E1 -10964.882,E2 -10964.882} C_VEL
LIN {X 0,Y 404.251,Z 300.127,A -85,B 0,C 180,E1 -10967.958,E2 -10967.958} C_VEL
LIN {X 0,Y 404.427,Z 300.104,A -85,B 0,C 180,E1 -10972.1,E2 -10972.1} C_VEL
LIN {X 0,Y 404.417,Z 300.107,A -85,B 0,C 180,E1 -10974.015,E2 -10974.015} C_VEL
LIN {X 0,Y 404.474,Z 300.101,A -85,B 0,C 180,E1 -10978.009,E2 -10978.009} C_VEL
LIN {X 0,Y 404.603,Z 300.085,A -85,B 0,C 180,E1 -10980,E2 -10980} C_VEL
LIN {X 0,Y 404.411,Z 300.105,A -85,B 0,C 180,E1 -10982.989,E2 -10982.989} C_VEL
LIN {X 0,Y 404.365,Z 300.112,A -85,B 0,C 180,E1 -10986.513,E2 -10986.513} C_VEL
LIN {X 0,Y 404.283,Z 300.121,A -85,B 0,C 180,E1 -10989.001,E2 -10989.001} C_VEL
LIN {X 0,Y 404.251,Z 300.133,A -85,B 0,C 180,E1 -10992.042,E2 -10992.042} C_VEL
LIN {X 0,Y 404.2,Z 300.131,A -85,B 0,C 180,E1 -10995.119,E2 -10995.119} C_VEL
LIN {X 0,Y 404.203,Z 300.139,A -85,B 0,C 180,E1 -10998.239,E2 -10998.239} C_VEL
LIN {X 0,Y 404.133,Z 300.14,A -85,B 0,C 180,E1 -11001.42,E2 -11001.42} C_VEL
LIN {X 0,Y 404.16,Z 300.141,A -85,B 0,C 180,E1 -11004.667,E2 -11004.667} C_VEL
LIN {X 0,Y 404.126,Z 300.143,A -85,B 0,C 180,E1 -11008.005,E2 -11008.005} C_VEL
LIN {X 0,Y 404.14,Z 300.143,A -85,B 0,C 180,E1 -11010.286,E2 -11010.286} C_VEL
LIN {X 0,Y 404.142,Z 300.139,A -85,B 0,C 180,E1 -11013.813,E2 -11013.813} C_VEL
LIN {X 0,Y 404.132,Z 300.146,A -85,B 0,C 180,E1 -11016.876,E2 -11016.876} C_VEL
LIN {X 0,Y 404.145,Z 300.139,A -85,B 0,C 180,E1 -11020.081,E2 -11020.081} C_VEL
LIN {X 0,Y 404.148,Z 300.143,A -85,B 0,C 180,E1 -11023.084,E2 -11023.084} C_VEL
LIN {X 0,Y 404.143,Z 300.138,A -85,B 0,C 180,E1 -11025.927,E2 -11025.927} C_VEL
LIN {X 0,Y 404.104,Z 300.146,A -85,B 0,C 180,E1 -11028.634,E2 -11028.634} C_VEL
LIN {X 0,Y 404.141,Z 300.142,A -85,B 0,C 180,E1 -11031.495,E2 -11031.495} C_VEL
LIN {X 0,Y 404.183,Z 300.138,A -85,B 0,C 180,E1 -11034.985,E2 -11034.985} C_VEL
LIN {X 0,Y 404.139,Z 300.139,A -85,B 0,C 180,E1 -11038.443,E2 -11038.443} C_VEL
LIN {X 0,Y 404.152,Z 300.139,A -85,B 0,C 180,E1 -11040.863,E2 -11040.863} C_VEL
LIN {X 0,Y 404.155,Z 300.138,A -85,B 0,C 180,E1 -11044.723,E2 -11044.723} C_VEL
LIN {X 0,Y 404.168,Z 300.143,A -85,B 0,C 180,E1 -11047.509,E2 -11047.509} C_VEL
LIN {X 0,Y 404.164,Z 300.136,A -85,B 0,C 180,E1 -11050.708,E2 -11050.708} C_VEL
LIN {X 0,Y 404.222,Z 300.135,A -85,B 0,C 180,E1 -11053.849,E2 -11053.849} C_VEL
LIN {X 0,Y 404.287,Z 300.121,A -85,B 0,C 180,E1 -11056.94,E2 -11056.94} C_VEL
LIN {X 0,Y 404.246,Z 300.132,A -85,B 0,C 180,E1 -11059.989,E2 -11059.989} C_VEL
LIN {X 0,Y 404.344,Z 300.113,A -85,B 0,C 180,E1 -11063.012,E2 -11063.012} C_VEL
LIN {X 0,Y 404.258,Z 300.124,A -85,B 0,C 180,E1 -11065.014,E2 -11065.014} C_VEL
LIN {X 0,Y 404.47,Z 300.104,A -85,B 0,C 180,E1 -11068.009,E2 -11068.009} C_VEL
LIN {X 0,Y 404.351,Z 300.113,A -85,B 0,C 180,E1 -11070.996,E2 -11070.996} C_VEL
LIN {X 0,Y 404.351,Z 300.113,A -85,B 0,C 180,E1 -11072.989,E2 -11072.989} C_VEL
LIN {X 0,Y 404.371,Z 300.114,A -85,B 0,C 180,E1 -11075.986,E2 -11075.986} C_VEL
LIN {X 0,Y 404.257,Z 300.126,A -85,B 0,C 180,E1 -11079.002,E2 -11079.002} C_VEL
LIN {X 0,Y 404.245,Z 300.128,A -85,B 0,C 180,E1 -11082.042,E2 -11082.042} C_VEL
LIN {X 0,Y 404.161,Z 300.138,A -85,B 0,C 180,E1 -11085.12,E2 -11085.12} C_VEL
LIN {X 0,Y 404.156,Z 300.139,A -85,B 0,C 180,E1 -11088.241,E2 -11088.241} C_VEL
LIN {X 0,Y 404.135,Z 300.144,A -85,B 0,C 180,E1 -11091.42,E2 -11091.42} C_VEL
LIN {X 0,Y 404.132,Z 300.143,A -85,B 0,C 180,E1 -11091.902,E2 -11091.902} C_VEL
LIN {X 0,Y 403.461,Z 300.24,A -85,B 0,C 180,E1 -11092.472,E2 -11092.472} C_VEL
LIN {X 0,Y 400.026,Z 300.755,A -85,B 0,C 180,E1 -11093.54,E2 -11093.54} C_VEL
LIN {X 0,Y 398.018,Z 301.965,A -85,B 0,C 180,E1 -11094.239,E2 -11094.239} C_VEL
LIN {X 0,Y 397.625,Z 303.559,A -85,B 0,C 180,E1 -11094.759,E2 -11094.759} C_VEL
LIN {X 0,Y 399.14,Z 312.249,A -85,B 0,C 180,E1 -11096.963,E2 -11096.963} C_VEL
LIN {X 0,Y 399.124,Z 313.569,A -85,B 0,C 180,E1 -11097.247,E2 -11097.247} C_VEL
LIN {X 0,Y 403.347,Z 335.755,A -85,B 0,C 180,E1 -11097.888,E2 -11097.888} C_VEL
LIN {X 0,Y 401.929,Z 421.14,A -85,B 0,C 180,E1 -11099.53,E2 -11099.53} C_VEL
LIN {X 0,Y 401.426,Z 434.834,A -85,B 0,C 180,E1 -11100.004,E2 -11100.004} C_VEL
LIN {X 0,Y 401.011,Z 446.808,A -85,B 0,C 180,E1 -11100.619,E2 -11100.619} C_VEL
LIN {X 0,Y 400.327,Z 458.189,A -85,B 0,C 180,E1 -11101.392,E2 -11101.392} C_VEL
LIN {X 0,Y 399.548,Z 469.725,A -85,B 0,C 180,E1 -11102.4,E2 -11102.4} C_VEL
LIN {X 0,Y 398.895,Z 480.271,A -85,B 0,C 180,E1 -11103.559,E2 -11103.559} C_VEL
LIN {X 0,Y 398.104,Z 489.809,A -85,B 0,C 180,E1 -11104.858,E2 -11104.858} C_VEL
LIN {X 0,Y 397.388,Z 498.55,A -85,B 0,C 180,E1 -11106.332,E2 -11106.332} C_VEL
LIN {X 0,Y 396.873,Z 505.235,A -85,B 0,C 180,E1 -11107.721,E2 -11107.721} C_VEL
LIN {X 0,Y 396.459,Z 510.933,A -85,B 0,C 180,E1 -11109.178,E2 -11109.178} C_VEL
LIN {X 0,Y 396.153,Z 516.522,A -85,B 0,C 180,E1 -11111.027,E2 -11111.027} C_VEL
LIN {X 0,Y 395.934,Z 519.684,A -85,B 0,C 180,E1 -11112.417,E2 -11112.417} C_VEL
LIN {X 0,Y 395.741,Z 522.019,A -85,B 0,C 180,E1 -11113.837,E2 -11113.837} C_VEL
LIN {X 0,Y 395.651,Z 523.548,A -85,B 0,C 180,E1 -11115.278,E2 -11115.278} C_VEL
LIN {X 0,Y 395.641,Z 524.275,A -85,B 0,C 180,E1 -11116.745,E2 -11116.745} C_VEL
LIN {X 0,Y 395.65,Z 524.158,A -85,B 0,C 180,E1 -11118.25,E2 -11118.25} C_VEL
LIN {X 0,Y 395.733,Z 522.619,A -85,B 0,C 180,E1 -11120.257,E2 -11120.257} C_VEL
LIN {X 0,Y 395.947,Z 520.694,A -85,B 0,C 180,E1 -11121.592,E2 -11121.592} C_VEL
LIN {X 0,Y 396.295,Z 516.469,A -85,B 0,C 180,E1 -11123.581,E2 -11123.581} C_VEL
LIN {X 0,Y 396.79,Z 510.679,A -85,B 0,C 180,E1 -11125.473,E2 -11125.473} C_VEL
LIN {X 0,Y 397.33,Z 504.411,A -85,B 0,C 180,E1 -11127.049,E2 -11127.049} C_VEL
LIN {X 0,Y 398.041,Z 496.545,A -85,B 0,C 180,E1 -11128.623,E2 -11128.623} C_VEL
LIN {X 0,Y 398.83,Z 488.204,A -85,B 0,C 180,E1 -11129.961,E2 -11129.961} C_VEL
LIN {X 0,Y 399.688,Z 477.518,A -85,B 0,C 180,E1 -11131.352,E2 -11131.352} C_VEL
LIN {X 0,Y 400.541,Z 467.046,A -85,B 0,C 180,E1 -11132.433,E2 -11132.433} C_VEL
LIN {X 0,Y 401.373,Z 455.278,A -85,B 0,C 180,E1 -11133.392,E2 -11133.392} C_VEL
LIN {X 0,Y 402.09,Z 443.099,A -85,B 0,C 180,E1 -11134.156,E2 -11134.156} C_VEL
LIN {X 0,Y 402.581,Z 429.966,A -85,B 0,C 180,E1 -11134.746,E2 -11134.746} C_VEL
LIN {X 0,Y 403.027,Z 416.275,A -85,B 0,C 180,E1 -11135.131,E2 -11135.131} C_VEL
LIN {X 0,Y 404.542,Z 334.807,A -85,B 0,C 180,E1 -11136.719,E2 -11136.719} C_VEL
LIN {X 0,Y 400.178,Z 314.563,A -85,B 0,C 180,E1 -11137.407,E2 -11137.407} C_VEL
LIN {X 0,Y 399.796,Z 313.03,A -85,B 0,C 180,E1 -11137.487,E2 -11137.487} C_VEL
LIN {X 0,Y 397.144,Z 301.017,A -85,B 0,C 180,E1 -11140.155,E2 -11140.155} C_VEL
LIN {X 0,Y 397.169,Z 301.019,A -85,B 0,C 180,E1 -11143.553,E2 -11143.553} C_VEL
LIN {X 0,Y 397.231,Z 301.006,A -85,B 0,C 180,E1 -11146.702,E2 -11146.702} C_VEL
LIN {X 0,Y 397.219,Z 301.006,A -85,B 0,C 180,E1 -11149.809,E2 -11149.809} C_VEL
LIN {X 0,Y 397.364,Z 300.987,A -85,B 0,C 180,E1 -11152.888,E2 -11152.888} C_VEL
LIN {X 0,Y 397.254,Z 301.001,A -85,B 0,C 180,E1 -11154.925,E2 -11154.925} C_VEL
LIN {X 0,Y 397.451,Z 300.976,A -85,B 0,C 180,E1 -11157.973,E2 -11157.973} C_VEL
LIN {X 0,Y 397.581,Z 300.961,A -85,B 0,C 180,E1 -11160,E2 -11160} C_VEL
LIN {X 0,Y 397.377,Z 300.983,A -85,B 0,C 180,E1 -11163.041,E2 -11163.041} C_VEL
LIN {X 0,Y 397.357,Z 300.988,A -85,B 0,C 180,E1 -11166.092,E2 -11166.092} C_VEL
LIN {X 0,Y 397.253,Z 300.998,A -85,B 0,C 180,E1 -11169.162,E2 -11169.162} C_VEL
LIN {X 0,Y 397.221,Z 301.007,A -85,B 0,C 180,E1 -11172.258,E2 -11172.258} C_VEL
LIN {X 0,Y 397.181,Z 301.008,A -85,B 0,C 180,E1 -11175.392,E2 -11175.392} C_VEL
LIN {X 0,Y 397.16,Z 301.014,A -85,B 0,C 180,E1 -11178.573,E2 -11178.573} C_VEL
LIN {X 0,Y 397.097,Z 301.015,A -85,B 0,C 180,E1 -11181.818,E2 -11181.818} C_VEL
LIN {X 0,Y 397.154,Z 301.01,A -85,B 0,C 180,E1 -11185.512,E2 -11185.512} C_VEL
LIN {X 0,Y 397.123,Z 301.011,A -85,B 0,C 180,E1 -11188.543,E2 -11188.543} C_VEL
LIN {X 0,Y 397.079,Z 301.017,A -85,B 0,C 180,E1 -11192.071,E2 -11192.071} C_VEL
LIN {X 0,Y 397.12,Z 301.018,A -85,B 0,C 180,E1 -11195.503,E2 -11195.503} C_VEL
LIN {X 0,Y 397.13,Z 301.015,A -85,B 0,C 180,E1 -11198.861,E2 -11198.861} C_VEL
LIN {X 0,Y 397.07,Z 301.023,A -85,B 0,C 180,E1 -11202.267,E2 -11202.267} C_VEL
LIN {X 0,Y 397.089,Z 301.024,A -85,B 0,C 180,E1 -11205.069,E2 -11205.069} C_VEL
LIN {X 0,Y 397.068,Z 301.023,A -85,B 0,C 180,E1 -11208.021,E2 -11208.021} C_VEL
LIN {X 0,Y 397.128,Z 301.018,A -85,B 0,C 180,E1 -11211.139,E2 -11211.139} C_VEL
LIN {X 0,Y 397.121,Z 301.021,A -85,B 0,C 180,E1 -11214.496,E2 -11214.496} C_VEL
LIN {X 0,Y 397.081,Z 301.029,A -85,B 0,C 180,E1 -11217.928,E2 -11217.928} C_VEL
LIN {X 0,Y 397.201,Z 301.196,A -85,B 0,C 180,E1 -11221.514,E2 -11221.514} C_VEL
LIN {X 0,Y 399.801,Z 313.233,A -85,B 0,C 180,E1 -11224.21,E2 -11224.21} C_VEL
LIN {X 0,Y 400.563,Z 318.503,A -85,B 0,C 180,E1 -11225.339,E2 -11225.339} C_VEL
LIN {X 0,Y 399.318,Z 337.192,A -85,B 0,C 180,E1 -11229.029,E2 -11229.029} C_VEL
LIN {X 0,Y 399.164,Z 340.065,A -85,B 0,C 180,E1 -11229.558,E2 -11229.558} C_VEL
LIN {X 0,Y 402.892,Z 361.976,A -85,B 0,C 180,E1 -11230.236,E2 -11230.236} C_VEL
LIN {X 0,Y 404.071,Z 371.679,A -85,B 0,C 180,E1 -11230.504,E2 -11230.504} C_VEL
LIN {X 0,Y 402.643,Z 450.058,A -85,B 0,C 180,E1 -11232.05,E2 -11232.05} C_VEL
LIN {X 0,Y 402.018,Z 463.431,A -85,B 0,C 180,E1 -11232.514,E2 -11232.514} C_VEL
LIN {X 0,Y 401.278,Z 475.69,A -85,B 0,C 180,E1 -11233.137,E2 -11233.137} C_VEL
LIN {X 0,Y 400.413,Z 487.54,A -85,B 0,C 180,E1 -11233.952,E2 -11233.952} C_VEL
LIN {X 0,Y 399.504,Z 499.248,A -85,B 0,C 180,E1 -11234.986,E2 -11234.986} C_VEL
LIN {X 0,Y 398.678,Z 509.327,A -85,B 0,C 180,E1 -11236.099,E2 -11236.099} C_VEL
LIN {X 0,Y 397.808,Z 519.496,A -85,B 0,C 180,E1 -11237.501,E2 -11237.501} C_VEL
LIN {X 0,Y 396.968,Z 528.443,A -85,B 0,C 180,E1 -11239.028,E2 -11239.028} C_VEL
LIN {X 0,Y 396.447,Z 535.619,A -85,B 0,C 180,E1 -11240.562,E2 -11240.562} C_VEL
LIN {X 0,Y 396.182,Z 540.506,A -85,B 0,C 180,E1 -11241.841,E2 -11241.841} C_VEL
LIN {X 0,Y 395.921,Z 545.236,A -85,B 0,C 180,E1 -11243.374,E2 -11243.374} C_VEL
LIN {X 0,Y 395.843,Z 548.847,A -85,B 0,C 180,E1 -11244.906,E2 -11244.906} C_VEL
LIN {X 0,Y 395.776,Z 550.672,A -85,B 0,C 180,E1 -11245.926,E2 -11245.926} C_VEL
LIN {X 0,Y 395.804,Z 553.052,A -85,B 0,C 180,E1 -11247.964,E2 -11247.964} C_VEL
LIN {X 0,Y 395.81,Z 553.639,A -85,B 0,C 180,E1 -11248.982,E2 -11248.982} C_VEL
LIN {X 0,Y 395.798,Z 553.777,A -85,B 0,C 180,E1 -11249.999,E2 -11249.999} C_VEL
LIN {X 0,Y 395.81,Z 553.512,A -85,B 0,C 180,E1 -11251.017,E2 -11251.017} C_VEL
LIN {X 0,Y 395.804,Z 552.85,A -85,B 0,C 180,E1 -11252.035,E2 -11252.035} C_VEL
LIN {X 0,Y 395.735,Z 551.778,A -85,B 0,C 180,E1 -11253.053,E2 -11253.053} C_VEL
LIN {X 0,Y 395.779,Z 550.243,A -85,B 0,C 180,E1 -11254.072,E2 -11254.072} C_VEL
LIN {X 0,Y 395.824,Z 546.638,A -85,B 0,C 180,E1 -11255.802,E2 -11255.802} C_VEL
LIN {X 0,Y 396.057,Z 541.285,A -85,B 0,C 180,E1 -11257.647,E2 -11257.647} C_VEL
LIN {X 0,Y 396.441,Z 534.314,A -85,B 0,C 180,E1 -11259.437,E2 -11259.437} C_VEL
LIN {X 0,Y 396.933,Z 526.742,A -85,B 0,C 180,E1 -11260.972,E2 -11260.972} C_VEL
LIN {X 0,Y 397.571,Z 519.016,A -85,B 0,C 180,E1 -11262.246,E2 -11262.246} C_VEL
LIN {X 0,Y 398.246,Z 510.085,A -85,B 0,C 180,E1 -11263.464,E2 -11263.464} C_VEL
LIN {X 0,Y 399.014,Z 499.142,A -85,B 0,C 180,E1 -11264.666,E2 -11264.666} C_VEL
LIN {X 0,Y 399.797,Z 487.536,A -85,B 0,C 180,E1 -11265.68,E2 -11265.68} C_VEL
LIN {X 0,Y 400.611,Z 475.327,A -85,B 0,C 180,E1 -11266.497,E2 -11266.497} C_VEL
LIN {X 0,Y 401.292,Z 461.819,A -85,B 0,C 180,E1 -11267.156,E2 -11267.156} C_VEL
LIN {X 0,Y 401.821,Z 449.397,A -85,B 0,C 180,E1 -11267.56,E2 -11267.56} C_VEL
LIN {X 0,Y 402.899,Z 369.458,A -85,B 0,C 180,E1 -11269.1,E2 -11269.1} C_VEL
LIN {X 0,Y 398.78,Z 341.442,A -85,B 0,C 180,E1 -11269.864,E2 -11269.864} C_VEL
LIN {X 0,Y 399.991,Z 324.768,A -85,B 0,C 180,E1 -11273.286,E2 -11273.286} C_VEL
LIN {X 0,Y 400.47,Z 318.135,A -85,B 0,C 180,E1 -11274.665,E2 -11274.665} C_VEL
LIN {X 0,Y 398.574,Z 307.717,A -85,B 0,C 180,E1 -11277.002,E2 -11277.002} C_VEL
LIN {X 0,Y 397.169,Z 301.012,A -85,B 0,C 180,E1 -11278.611,E2 -11278.611} C_VEL
LIN {X 0,Y 397.077,Z 301.026,A -85,B 0,C 180,E1 -11282.071,E2 -11282.071} C_VEL
LIN {X 0,Y 397.117,Z 301.014,A -85,B 0,C 180,E1 -11285.503,E2 -11285.503} C_VEL
LIN {X 0,Y 397.123,Z 301.015,A -85,B 0,C 180,E1 -11288.86,E2 -11288.86} C_VEL
LIN {X 0,Y 397.065,Z 301.026,A -85,B 0,C 180,E1 -11292.266,E2 -11292.266} C_VEL
LIN {X 0,Y 397.086,Z 301.019,A -85,B 0,C 180,E1 -11295.068,E2 -11295.068} C_VEL
LIN {X 0,Y 397.065,Z 301.022,A -85,B 0,C 180,E1 -11298.02,E2 -11298.02} C_VEL
LIN {X 0,Y 397.129,Z 301.014,A -85,B 0,C 180,E1 -11301.137,E2 -11301.137} C_VEL
LIN {X 0,Y 397.115,Z 301.018,A -85,B 0,C 180,E1 -11304.496,E2 -11304.496} C_VEL
LIN {X 0,Y 397.073,Z 301.019,A -85,B 0,C 180,E1 -11307.928,E2 -11307.928} C_VEL
LIN {X 0,Y 397.116,Z 301.016,A -85,B 0,C 180,E1 -11311.456,E2 -11311.456} C_VEL
LIN {X 0,Y 397.147,Z 301.012,A -85,B 0,C 180,E1 -11314.487,E2 -11314.487} C_VEL
LIN {X 0,Y 397.104,Z 301.023,A -85,B 0,C 180,E1 -11317.085,E2 -11317.085} C_VEL
LIN {X 0,Y 397.142,Z 301.011,A -85,B 0,C 180,E1 -11320.353,E2 -11320.353} C_VEL
LIN {X 0,Y 397.161,Z 301.012,A -85,B 0,C 180,E1 -11323.553,E2 -11323.553} C_VEL
LIN {X 0,Y 397.223,Z 301.002,A -85,B 0,C 180,E1 -11326.703,E2 -11326.703} C_VEL
LIN {X 0,Y 397.212,Z 301.005,A -85,B 0,C 180,E1 -11329.809,E2 -11329.809} C_VEL
LIN {X 0,Y 397.358,Z 300.985,A -85,B 0,C 180,E1 -11332.888,E2 -11332.888} C_VEL
LIN {X 0,Y 397.248,Z 300.998,A -85,B 0,C 180,E1 -11334.925,E2 -11334.925} C_VEL
LIN {X 0,Y 397.443,Z 300.977,A -85,B 0,C 180,E1 -11337.973,E2 -11337.973} C_VEL
LIN {X 0,Y 397.572,Z 300.961,A -85,B 0,C 180,E1 -11340,E2 -11340} C_VEL
LIN {X 0,Y 397.371,Z 300.983,A -85,B 0,C 180,E1 -11343.042,E2 -11343.042} C_VEL
LIN {X 0,Y 397.319,Z 300.99,A -85,B 0,C 180,E1 -11346.506,E2 -11346.506} C_VEL
LIN {X 0,Y 397.246,Z 300.998,A -85,B 0,C 180,E1 -11349.162,E2 -11349.162} C_VEL
LIN {X 0,Y 397.214,Z 301.007,A -85,B 0,C 180,E1 -11352.259,E2 -11352.259} C_VEL
LIN {X 0,Y 397.173,Z 301.007,A -85,B 0,C 180,E1 -11355.393,E2 -11355.393} C_VEL
LIN {X 0,Y 397.156,Z 301.012,A -85,B 0,C 180,E1 -11358.574,E2 -11358.574} C_VEL
LIN {X 0,Y 397.091,Z 301.019,A -85,B 0,C 180,E1 -11361.819,E2 -11361.819} C_VEL
LIN {X 0,Y 397.118,Z 301.014,A -85,B 0,C 180,E1 -11365.135,E2 -11365.135} C_VEL
LIN {X 0,Y 397.076,Z 301.026,A -85,B 0,C 180,E1 -11368.548,E2 -11368.548} C_VEL
LIN {X 0,Y 397.078,Z 301.019,A -85,B 0,C 180,E1 -11371.837,E2 -11371.837} C_VEL
LIN {X 0,Y 397.122,Z 301.019,A -85,B 0,C 180,E1 -11374.494,E2 -11374.494} C_VEL
LIN {X 0,Y 397.095,Z 301.019,A -85,B 0,C 180,E1 -11378.277,E2 -11378.277} C_VEL
LIN {X 0,Y 397.083,Z 301.025,A -85,B 0,C 180,E1 -11380.91,E2 -11380.91} C_VEL
LIN {X 0,Y 397.098,Z 301.017,A -85,B 0,C 180,E1 -11383.65,E2 -11383.65} C_VEL
LIN {X 0,Y 397.096,Z 301.019,A -85,B 0,C 180,E1 -11386.523,E2 -11386.523} C_VEL
LIN {X 0,Y 397.086,Z 301.019,A -85,B 0,C 180,E1 -11390.421,E2 -11390.421} C_VEL
LIN {X 0,Y 397.097,Z 301.022,A -85,B 0,C 180,E1 -11393.006,E2 -11393.006} C_VEL
LIN {X 0,Y 397.118,Z 301.014,A -85,B 0,C 180,E1 -11396.283,E2 -11396.283} C_VEL
LIN {X 0,Y 397.099,Z 301.016,A -85,B 0,C 180,E1 -11400.138,E2 -11400.138} C_VEL
LIN {X 0,Y 397.078,Z 301.023,A -85,B 0,C 180,E1 -11403.738,E2 -11403.738} C_VEL
LIN {X 0,Y 397.1,Z 301.018,A -85,B 0,C 180,E1 -11407.086,E2 -11407.086} C_VEL
LIN {X 0,Y 397.149,Z 301.01,A -85,B 0,C 180,E1 -11410.354,E2 -11410.354} C_VEL
LIN {X 0,Y 397.168,Z 301.013,A -85,B 0,C 180,E1 -11413.554,E2 -11413.554} C_VEL
LIN {X 0,Y 397.232,Z 300.999,A -85,B 0,C 180,E1 -11416.704,E2 -11416.704} C_VEL
LIN {X 0,Y 397.207,Z 301.009,A -85,B 0,C 180,E1 -11419.809,E2 -11419.809} C_VEL
LIN {X 0,Y 397.297,Z 300.991,A -85,B 0,C 180,E1 -11422.888,E2 -11422.888} C_VEL
LIN {X 0,Y 397.23,Z 301,A -85,B 0,C 180,E1 -11424.925,E2 -11424.925} C_VEL
LIN {X 0,Y 397.437,Z 300.98,A -85,B 0,C 180,E1 -11427.974,E2 -11427.974} C_VEL
LIN {X 0,Y 397.321,Z 300.989,A -85,B 0,C 180,E1 -11431.014,E2 -11431.014} C_VEL
LIN {X 0,Y 397.287,Z 300.993,A -85,B 0,C 180,E1 -11433.043,E2 -11433.043} C_VEL
LIN {X 0,Y 397.324,Z 300.993,A -85,B 0,C 180,E1 -11436.093,E2 -11436.093} C_VEL
LIN {X 0,Y 397.228,Z 301,A -85,B 0,C 180,E1 -11439.163,E2 -11439.163} C_VEL
LIN {X 0,Y 397.208,Z 301.007,A -85,B 0,C 180,E1 -11442.259,E2 -11442.259} C_VEL
LIN {X 0,Y 397.114,Z 301.014,A -85,B 0,C 180,E1 -11445.395,E2 -11445.395} C_VEL
LIN {X 0,Y 397.124,Z 301.013,A -85,B 0,C 180,E1 -11447.509,E2 -11447.509} C_VEL
LIN {X 0,Y 397.099,Z 301.024,A -85,B 0,C 180,E1 -11450.731,E2 -11450.731} C_VEL
LIN {X 0,Y 397.156,Z 301.104,A -85,B 0,C 180,E1 -11454.121,E2 -11454.121} C_VEL
LIN {X 0,Y 397.625,Z 303.559,A -85,B 0,C 180,E1 -11454.759,E2 -11454.759} C_VEL
LIN {X 0,Y 397.32,Z 305.84,A -85,B 0,C 180,E1 -11455.3,E2 -11455.3} C_VEL
LIN {X 0,Y 394.973,Z 309.839,A -85,B 0,C 180,E1 -11456.144,E2 -11456.144} C_VEL
LIN {X 0,Y 393.099,Z 313.459,A -85,B 0,C 180,E1 -11456.743,E2 -11456.743} C_VEL
LIN {X 0,Y 392.765,Z 316.044,A -85,B 0,C 180,E1 -11456.977,E2 -11456.977} C_VEL
LIN {X 0,Y 392.902,Z 317.197,A -85,B 0,C 180,E1 -11457.029,E2 -11457.029} C_VEL
LIN {X 0,Y 396.585,Z 336.551,A -85,B 0,C 180,E1 -11457.598,E2 -11457.598} C_VEL
LIN {X 0,Y 395.105,Z 421.589,A -85,B 0,C 180,E1 -11459.27,E2 -11459.27} C_VEL
LIN {X 0,Y 394.557,Z 435.449,A -85,B 0,C 180,E1 -11459.761,E2 -11459.761} C_VEL
LIN {X 0,Y 394.105,Z 447.535,A -85,B 0,C 180,E1 -11460.399,E2 -11460.399} C_VEL
LIN {X 0,Y 393.31,Z 460.055,A -85,B 0,C 180,E1 -11461.287,E2 -11461.287} C_VEL
LIN {X 0,Y 392.527,Z 471.544,A -85,B 0,C 180,E1 -11462.337,E2 -11462.337} C_VEL
LIN {X 0,Y 391.845,Z 481.533,A -85,B 0,C 180,E1 -11463.486,E2 -11463.486} C_VEL
LIN {X 0,Y 391.039,Z 491.41,A -85,B 0,C 180,E1 -11464.893,E2 -11464.893} C_VEL
LIN {X 0,Y 390.258,Z 500.284,A -85,B 0,C 180,E1 -11466.462,E2 -11466.462} C_VEL
LIN {X 0,Y 389.669,Z 507.71,A -85,B 0,C 180,E1 -11468.132,E2 -11468.132} C_VEL
LIN {X 0,Y 389.263,Z 513.748,A -85,B 0,C 180,E1 -11469.862,E2 -11469.862} C_VEL
LIN {X 0,Y 389.033,Z 517.553,A -85,B 0,C 180,E1 -11471.27,E2 -11471.27} C_VEL
LIN {X 0,Y 388.785,Z 520.629,A -85,B 0,C 180,E1 -11472.754,E2 -11472.754} C_VEL
LIN {X 0,Y 388.668,Z 522.078,A -85,B 0,C 180,E1 -11473.672,E2 -11473.672} C_VEL
LIN {X 0,Y 388.566,Z 523.698,A -85,B 0,C 180,E1 -11475.138,E2 -11475.138} C_VEL
LIN {X 0,Y 388.562,Z 524.507,A -85,B 0,C 180,E1 -11476.581,E2 -11476.581} C_VEL
LIN {X 0,Y 388.565,Z 524.536,A -85,B 0,C 180,E1 -11477.992,E2 -11477.992} C_VEL
LIN {X 0,Y 388.583,Z 523.773,A -85,B 0,C 180,E1 -11479.431,E2 -11479.431} C_VEL
LIN {X 0,Y 388.768,Z 522.033,A -85,B 0,C 180,E1 -11481.018,E2 -11481.018} C_VEL
LIN {X 0,Y 389.033,Z 519.222,A -85,B 0,C 180,E1 -11482.644,E2 -11482.644} C_VEL
LIN {X 0,Y 389.4,Z 515.184,A -85,B 0,C 180,E1 -11484.309,E2 -11484.309} C_VEL
LIN {X 0,Y 389.925,Z 509.65,A -85,B 0,C 180,E1 -11486.031,E2 -11486.031} C_VEL
LIN {X 0,Y 390.568,Z 502.456,A -85,B 0,C 180,E1 -11487.751,E2 -11487.751} C_VEL
LIN {X 0,Y 391.405,Z 494.053,A -85,B 0,C 180,E1 -11489.344,E2 -11489.344} C_VEL
LIN {X 0,Y 392.322,Z 484.536,A -85,B 0,C 180,E1 -11490.78,E2 -11490.78} C_VEL
LIN {X 0,Y 393.145,Z 474.428,A -85,B 0,C 180,E1 -11492.014,E2 -11492.014} C_VEL
LIN {X 0,Y 394.083,Z 463.451,A -85,B 0,C 180,E1 -11493.087,E2 -11493.087} C_VEL
LIN {X 0,Y 394.837,Z 452.494,A -85,B 0,C 180,E1 -11493.932,E2 -11493.932} C_VEL
LIN {X 0,Y 395.536,Z 440.917,A -85,B 0,C 180,E1 -11494.617,E2 -11494.617} C_VEL
LIN {X 0,Y 395.994,Z 428.446,A -85,B 0,C 180,E1 -11495.157,E2 -11495.157} C_VEL
LIN {X 0,Y 396.409,Z 415.889,A -85,B 0,C 180,E1 -11495.499,E2 -11495.499} C_VEL
LIN {X 0,Y 397.901,Z 335.471,A -85,B 0,C 180,E1 -11497.099,E2 -11497.099} C_VEL
LIN {X 0,Y 393.697,Z 316.169,A -85,B 0,C 180,E1 -11497.781,E2 -11497.781} C_VEL
LIN {X 0,Y 392.678,Z 313.423,A -85,B 0,C 180,E1 -11497.923,E2 -11497.923} C_VEL
LIN {X 0,Y 390.118,Z 301.893,A -85,B 0,C 180,E1 -11500.532,E2 -11500.532} C_VEL
LIN {X 0,Y 390.141,Z 301.894,A -85,B 0,C 180,E1 -11503.248,E2 -11503.248} C_VEL
LIN {X 0,Y 390.197,Z 301.882,A -85,B 0,C 180,E1 -11506.561,E2 -11506.561} C_VEL
LIN {X 0,Y 390.207,Z 301.878,A -85,B 0,C 180,E1 -11510.671,E2 -11510.671} C_VEL
LIN {X 0,Y 390.319,Z 301.865,A -85,B 0,C 180,E1 -11512.759,E2 -11512.759} C_VEL
LIN {X 0,Y 390.226,Z 301.876,A -85,B 0,C 180,E1 -11514.833,E2 -11514.833} C_VEL
LIN {X 0,Y 390.419,Z 301.852,A -85,B 0,C 180,E1 -11517.937,E2 -11517.937} C_VEL
LIN {X 0,Y 390.55,Z 301.837,A -85,B 0,C 180,E1 -11520,E2 -11520} C_VEL
LIN {X 0,Y 390.311,Z 301.863,A -85,B 0,C 180,E1 -11523.096,E2 -11523.096} C_VEL
LIN {X 0,Y 390.309,Z 301.864,A -85,B 0,C 180,E1 -11526.202,E2 -11526.202} C_VEL
LIN {X 0,Y 390.205,Z 301.876,A -85,B 0,C 180,E1 -11529.329,E2 -11529.329} C_VEL
LIN {X 0,Y 390.196,Z 301.873,A -85,B 0,C 180,E1 -11533.438,E2 -11533.438} C_VEL
LIN {X 0,Y 390.13,Z 301.881,A -85,B 0,C 180,E1 -11537.298,E2 -11537.298} C_VEL
LIN {X 0,Y 390.089,Z 301.89,A -85,B 0,C 180,E1 -11540.47,E2 -11540.47} C_VEL
LIN {X 0,Y 390.075,Z 301.891,A -85,B 0,C 180,E1 -11543.352,E2 -11543.352} C_VEL
LIN {X 0,Y 390.115,Z 301.89,A -85,B 0,C 180,E1 -11546.768,E2 -11546.768} C_VEL
LIN {X 0,Y 390.041,Z 301.898,A -85,B 0,C 180,E1 -11550.3,E2 -11550.3} C_VEL
LIN {X 0,Y 390.07,Z 301.892,A -85,B 0,C 180,E1 -11554.024,E2 -11554.024} C_VEL
LIN {X 0,Y 390.044,Z 301.895,A -85,B 0,C 180,E1 -11557.55,E2 -11557.55} C_VEL
LIN {X 0,Y 390.058,Z 301.895,A -85,B 0,C 180,E1 -11560.821,E2 -11560.821} C_VEL
LIN {X 0,Y 390.056,Z 301.898,A -85,B 0,C 180,E1 -11563.886,E2 -11563.886} C_VEL
LIN {X 0,Y 390.059,Z 301.896,A -85,B 0,C 180,E1 -11566.789,E2 -11566.789} C_VEL
LIN {X 0,Y 390.058,Z 301.899,A -85,B 0,C 180,E1 -11569.56,E2 -11569.56} C_VEL
LIN {X 0,Y 390.044,Z 301.901,A -85,B 0,C 180,E1 -11572.449,E2 -11572.449} C_VEL
LIN {X 0,Y 390.07,Z 301.903,A -85,B 0,C 180,E1 -11575.975,E2 -11575.975} C_VEL
LIN {X 0,Y 390.049,Z 301.899,A -85,B 0,C 180,E1 -11579.869,E2 -11579.869} C_VEL
LIN {X 0,Y 390.123,Z 301.965,A -85,B 0,C 180,E1 -11581.124,E2 -11581.124} C_VEL
LIN {X 0,Y 392.639,Z 313.387,A -85,B 0,C 180,E1 -11583.745,E2 -11583.745} C_VEL
LIN {X 0,Y 393.683,Z 319.986,A -85,B 0,C 180,E1 -11585.196,E2 -11585.196} C_VEL
LIN {X 0,Y 392.488,Z 336.987,A -85,B 0,C 180,E1 -11588.611,E2 -11588.611} C_VEL
LIN {X 0,Y 392.31,Z 339.759,A -85,B 0,C 180,E1 -11589.127,E2 -11589.127} C_VEL
LIN {X 0,Y 396.075,Z 361.17,A -85,B 0,C 180,E1 -11589.822,E2 -11589.822} C_VEL
LIN {X 0,Y 397.48,Z 372.312,A -85,B 0,C 180,E1 -11590.14,E2 -11590.14} C_VEL
LIN {X 0,Y 395.962,Z 449.849,A -85,B 0,C 180,E1 -11591.703,E2 -11591.703} C_VEL
LIN {X 0,Y 395.302,Z 463.15,A -85,B 0,C 180,E1 -11592.173,E2 -11592.173} C_VEL
LIN {X 0,Y 394.519,Z 475.878,A -85,B 0,C 180,E1 -11592.839,E2 -11592.839} C_VEL
LIN {X 0,Y 393.611,Z 487.602,A -85,B 0,C 180,E1 -11593.667,E2 -11593.667} C_VEL
LIN {X 0,Y 392.664,Z 498.99,A -85,B 0,C 180,E1 -11594.692,E2 -11594.692} C_VEL
LIN {X 0,Y 391.722,Z 509.795,A -85,B 0,C 180,E1 -11595.917,E2 -11595.917} C_VEL
LIN {X 0,Y 390.865,Z 519.402,A -85,B 0,C 180,E1 -11597.275,E2 -11597.275} C_VEL
LIN {X 0,Y 389.979,Z 528.325,A -85,B 0,C 180,E1 -11598.829,E2 -11598.829} C_VEL
LIN {X 0,Y 389.418,Z 535.464,A -85,B 0,C 180,E1 -11600.39,E2 -11600.39} C_VEL
LIN {X 0,Y 389.02,Z 542.016,A -85,B 0,C 180,E1 -11602.212,E2 -11602.212} C_VEL
LIN {X 0,Y 388.774,Z 546.54,A -85,B 0,C 180,E1 -11603.855,E2 -11603.855} C_VEL
LIN {X 0,Y 388.74,Z 548.637,A -85,B 0,C 180,E1 -11604.813,E2 -11604.813} C_VEL
LIN {X 0,Y 388.701,Z 550.444,A -85,B 0,C 180,E1 -11605.852,E2 -11605.852} C_VEL
LIN {X 0,Y 388.701,Z 552.806,A -85,B 0,C 180,E1 -11607.927,E2 -11607.927} C_VEL
LIN {X 0,Y 388.739,Z 553.381,A -85,B 0,C 180,E1 -11608.963,E2 -11608.963} C_VEL
LIN {X 0,Y 388.727,Z 553.508,A -85,B 0,C 180,E1 -11609.999,E2 -11609.999} C_VEL
LIN {X 0,Y 388.739,Z 553.234,A -85,B 0,C 180,E1 -11611.035,E2 -11611.035} C_VEL
LIN {X 0,Y 388.703,Z 552.562,A -85,B 0,C 180,E1 -11612.072,E2 -11612.072} C_VEL
LIN {X 0,Y 388.642,Z 551.474,A -85,B 0,C 180,E1 -11613.109,E2 -11613.109} C_VEL
LIN {X 0,Y 388.704,Z 549.925,A -85,B 0,C 180,E1 -11614.147,E2 -11614.147} C_VEL
LIN {X 0,Y 388.725,Z 546.675,A -85,B 0,C 180,E1 -11615.752,E2 -11615.752} C_VEL
LIN {X 0,Y 388.93,Z 542.559,A -85,B 0,C 180,E1 -11617.266,E2 -11617.266} C_VEL
LIN {X 0,Y 389.244,Z 536.098,A -85,B 0,C 180,E1 -11619.089,E2 -11619.089} C_VEL
LIN {X 0,Y 389.696,Z 529.034,A -85,B 0,C 180,E1 -11620.652,E2 -11620.652} C_VEL
LIN {X 0,Y 390.446,Z 520.167,A -85,B 0,C 180,E1 -11622.21,E2 -11622.21} C_VEL
LIN {X 0,Y 391.173,Z 511.076,A -85,B 0,C 180,E1 -11623.506,E2 -11623.506} C_VEL
LIN {X 0,Y 391.941,Z 501.07,A -85,B 0,C 180,E1 -11624.671,E2 -11624.671} C_VEL
LIN {X 0,Y 392.703,Z 489.958,A -85,B 0,C 180,E1 -11625.704,E2 -11625.704} C_VEL
LIN {X 0,Y 393.569,Z 477.55,A -85,B 0,C 180,E1 -11626.601,E2 -11626.601} C_VEL
LIN {X 0,Y 394.242,Z 465.823,A -85,B 0,C 180,E1 -11627.239,E2 -11627.239} C_VEL
LIN {X 0,Y 394.818,Z 453.292,A -85,B 0,C 180,E1 -11627.714,E2 -11627.714} C_VEL
LIN {X 0,Y 395.191,Z 436.212,A -85,B 0,C 180,E1 -11628.098,E2 -11628.098} C_VEL
LIN {X 0,Y 396.069,Z 369.813,A -85,B 0,C 180,E1 -11629.393,E2 -11629.393} C_VEL
LIN {X 0,Y 391.864,Z 341.183,A -85,B 0,C 180,E1 -11630.196,E2 -11630.196} C_VEL
LIN {X 0,Y 393.271,Z 323.058,A -85,B 0,C 180,E1 -11633.988,E2 -11633.988} C_VEL
LIN {X 0,Y 393.492,Z 319.155,A -85,B 0,C 180,E1 -11634.816,E2 -11634.816} C_VEL
LIN {X 0,Y 391.544,Z 308.585,A -85,B 0,C 180,E1 -11637.239,E2 -11637.239} C_VEL
LIN {X 0,Y 390.12,Z 301.889,A -85,B 0,C 180,E1 -11638.843,E2 -11638.843} C_VEL
LIN {X 0,Y 390.041,Z 301.901,A -85,B 0,C 180,E1 -11642.721,E2 -11642.721} C_VEL
LIN {X 0,Y 390.053,Z 301.896,A -85,B 0,C 180,E1 -11645.825,E2 -11645.825} C_VEL
LIN {X 0,Y 390.064,Z 301.893,A -85,B 0,C 180,E1 -11649.217,E2 -11649.217} C_VEL
LIN {X 0,Y 390.039,Z 301.903,A -85,B 0,C 180,E1 -11652.374,E2 -11652.374} C_VEL
LIN {X 0,Y 390.043,Z 301.895,A -85,B 0,C 180,E1 -11655.354,E2 -11655.354} C_VEL
LIN {X 0,Y 390.029,Z 301.9,A -85,B 0,C 180,E1 -11658.186,E2 -11658.186} C_VEL
LIN {X 0,Y 390.088,Z 301.894,A -85,B 0,C 180,E1 -11660.907,E2 -11660.907} C_VEL
LIN {X 0,Y 390.081,Z 301.898,A -85,B 0,C 180,E1 -11664.793,E2 -11664.793} C_VEL
LIN {X 0,Y 390.019,Z 301.901,A -85,B 0,C 180,E1 -11668.495,E2 -11668.495} C_VEL
LIN {X 0,Y 390.112,Z 301.887,A -85,B 0,C 180,E1 -11672.07,E2 -11672.07} C_VEL
LIN {X 0,Y 390.074,Z 301.893,A -85,B 0,C 180,E1 -11675.519,E2 -11675.519} C_VEL
LIN {X 0,Y 390.05,Z 301.898,A -85,B 0,C 180,E1 -11678.878,E2 -11678.878} C_VEL
LIN {X 0,Y 390.122,Z 301.885,A -85,B 0,C 180,E1 -11682.167,E2 -11682.167} C_VEL
LIN {X 0,Y 390.138,Z 301.89,A -85,B 0,C 180,E1 -11685.393,E2 -11685.393} C_VEL
LIN {X 0,Y 390.142,Z 301.883,A -85,B 0,C 180,E1 -11688.571,E2 -11688.571} C_VEL
LIN {X 0,Y 390.338,Z 301.86,A -85,B 0,C 180,E1 -11691.993,E2 -11691.993} C_VEL
LIN {X 0,Y 390.22,Z 301.873,A -85,B 0,C 180,E1 -11694.834,E2 -11694.834} C_VEL
LIN {X 0,Y 390.412,Z 301.853,A -85,B 0,C 180,E1 -11697.937,E2 -11697.937} C_VEL
LIN {X 0,Y 390.542,Z 301.837,A -85,B 0,C 180,E1 -11700,E2 -11700} C_VEL
LIN {X 0,Y 390.305,Z 301.863,A -85,B 0,C 180,E1 -11703.097,E2 -11703.097} C_VEL
LIN {X 0,Y 390.278,Z 301.867,A -85,B 0,C 180,E1 -11706.496,E2 -11706.496} C_VEL
LIN {X 0,Y 390.198,Z 301.877,A -85,B 0,C 180,E1 -11709.329,E2 -11709.329} C_VEL
LIN {X 0,Y 390.189,Z 301.878,A -85,B 0,C 180,E1 -11713.439,E2 -11713.439} C_VEL
LIN {X 0,Y 390.144,Z 301.883,A -85,B 0,C 180,E1 -11717.308,E2 -11717.308} C_VEL
LIN {X 0,Y 390.082,Z 301.895,A -85,B 0,C 180,E1 -11720.471,E2 -11720.471} C_VEL
LIN {X 0,Y 390.061,Z 301.893,A -85,B 0,C 180,E1 -11723.353,E2 -11723.353} C_VEL
LIN {X 0,Y 390.051,Z 301.898,A -85,B 0,C 180,E1 -11726.773,E2 -11726.773} C_VEL
LIN {X 0,Y 390.033,Z 301.901,A -85,B 0,C 180,E1 -11730.301,E2 -11730.301} C_VEL
LIN {X 0,Y 390.065,Z 301.893,A -85,B 0,C 180,E1 -11734.025,E2 -11734.025} C_VEL
LIN {X 0,Y 390.038,Z 301.896,A -85,B 0,C 180,E1 -11737.551,E2 -11737.551} C_VEL
LIN {X 0,Y 390.051,Z 301.902,A -85,B 0,C 180,E1 -11740.822,E2 -11740.822} C_VEL
LIN {X 0,Y 390.052,Z 301.894,A -85,B 0,C 180,E1 -11743.887,E2 -11743.887} C_VEL
LIN {X 0,Y 390.05,Z 301.899,A -85,B 0,C 180,E1 -11746.79,E2 -11746.79} C_VEL
LIN {X 0,Y 390.009,Z 301.901,A -85,B 0,C 180,E1 -11749.556,E2 -11749.556} C_VEL
LIN {X 0,Y 390.04,Z 301.896,A -85,B 0,C 180,E1 -11752.451,E2 -11752.451} C_VEL
LIN {X 0,Y 390.068,Z 301.892,A -85,B 0,C 180,E1 -11755.976,E2 -11755.976} C_VEL
LIN {X 0,Y 390.044,Z 301.897,A -85,B 0,C 180,E1 -11759.871,E2 -11759.871} C_VEL
LIN {X 0,Y 390.032,Z 301.901,A -85,B 0,C 180,E1 -11763.227,E2 -11763.227} C_VEL
LIN {X 0,Y 390.066,Z 301.893,A -85,B 0,C 180,E1 -11766.766,E2 -11766.766} C_VEL
LIN {X 0,Y 390.109,Z 301.89,A -85,B 0,C 180,E1 -11769.984,E2 -11769.984} C_VEL
LIN {X 0,Y 390.14,Z 301.885,A -85,B 0,C 180,E1 -11773.249,E2 -11773.249} C_VEL
LIN {X 0,Y 390.198,Z 301.876,A -85,B 0,C 180,E1 -11776.562,E2 -11776.562} C_VEL
LIN {X 0,Y 390.188,Z 301.877,A -85,B 0,C 180,E1 -11780.672,E2 -11780.672} C_VEL
LIN {X 0,Y 390.279,Z 301.871,A -85,B 0,C 180,E1 -11783.798,E2 -11783.798} C_VEL
LIN {X 0,Y 390.403,Z 301.855,A -85,B 0,C 180,E1 -11787.937,E2 -11787.937} C_VEL
LIN {X 0,Y 390.292,Z 301.864,A -85,B 0,C 180,E1 -11791.032,E2 -11791.032} C_VEL
LIN {X 0,Y 390.402,Z 301.856,A -85,B 0,C 180,E1 -11792.064,E2 -11792.064} C_VEL
LIN {X 0,Y 390.279,Z 301.871,A -85,B 0,C 180,E1 -11796.203,E2 -11796.203} C_VEL
LIN {X 0,Y 390.187,Z 301.877,A -85,B 0,C 180,E1 -11799.33,E2 -11799.33} C_VEL
LIN {X 0,Y 390.156,Z 301.888,A -85,B 0,C 180,E1 -11802.484,E2 -11802.484} C_VEL
LIN {X 0,Y 390.06,Z 301.893,A -85,B 0,C 180,E1 -11805.681,E2 -11805.681} C_VEL
LIN {X 0,Y 390.066,Z 301.892,A -85,B 0,C 180,E1 -11807.837,E2 -11807.837} C_VEL
LIN {X 0,Y 390.054,Z 301.899,A -85,B 0,C 180,E1 -11811.123,E2 -11811.123} C_VEL
LIN {X 0,Y 390.139,Z 302.043,A -85,B 0,C 180,E1 -11813.911,E2 -11813.911} C_VEL
LIN {X 0,Y 392.195,Z 313.577,A -85,B 0,C 180,E1 -11816.903,E2 -11816.903} C_VEL
LIN {X 0,Y 392.902,Z 317.197,A -85,B 0,C 180,E1 -11817.029,E2 -11817.029} C_VEL
LIN {X 0,Y 393.368,Z 323.022,A -85,B 0,C 180,E1 -11817.172,E2 -11817.172} C_VEL
LIN {X 0,Y 392.794,Z 328.926,A -85,B 0,C 180,E1 -11817.266,E2 -11817.266} C_VEL
LIN {X 0,Y 389.868,Z 344.735,A -85,B 0,C 180,E1 -11817.455,E2 -11817.455} C_VEL
LIN {X 0,Y 389.606,Z 348.731,A -85,B 0,C 180,E1 -11817.525,E2 -11817.525} C_VEL
LIN {X 0,Y 388.261,Z 421.981,A -85,B 0,C 180,E1 -11818.998,E2 -11818.998} C_VEL
LIN {X 0,Y 387.711,Z 435.944,A -85,B 0,C 180,E1 -11819.506,E2 -11819.506} C_VEL
LIN {X 0,Y 387.205,Z 448.365,A -85,B 0,C 180,E1 -11820.181,E2 -11820.181} C_VEL
LIN {X 0,Y 386.384,Z 460.827,A -85,B 0,C 180,E1 -11821.09,E2 -11821.09} C_VEL
LIN {X 0,Y 385.629,Z 471.248,A -85,B 0,C 180,E1 -11822.06,E2 -11822.06} C_VEL
LIN {X 0,Y 384.943,Z 481.23,A -85,B 0,C 180,E1 -11823.211,E2 -11823.211} C_VEL
LIN {X 0,Y 384.118,Z 490.812,A -85,B 0,C 180,E1 -11824.578,E2 -11824.578} C_VEL
LIN {X 0,Y 383.42,Z 498.484,A -85,B 0,C 180,E1 -11825.913,E2 -11825.913} C_VEL
LIN {X 0,Y 382.771,Z 506.173,A -85,B 0,C 180,E1 -11827.56,E2 -11827.56} C_VEL
LIN {X 0,Y 382.263,Z 513.005,A -85,B 0,C 180,E1 -11829.449,E2 -11829.449} C_VEL
LIN {X 0,Y 381.977,Z 517.394,A -85,B 0,C 180,E1 -11831.03,E2 -11831.03} C_VEL
LIN {X 0,Y 381.672,Z 521.291,A -85,B 0,C 180,E1 -11832.946,E2 -11832.946} C_VEL
LIN {X 0,Y 381.494,Z 523.294,A -85,B 0,C 180,E1 -11834.431,E2 -11834.431} C_VEL
LIN {X 0,Y 381.448,Z 524.494,A -85,B 0,C 180,E1 -11835.936,E2 -11835.936} C_VEL
LIN {X 0,Y 381.454,Z 524.878,A -85,B 0,C 180,E1 -11837.474,E2 -11837.474} C_VEL
LIN {X 0,Y 381.483,Z 524.381,A -85,B 0,C 180,E1 -11839.055,E2 -11839.055} C_VEL
LIN {X 0,Y 381.619,Z 522.924,A -85,B 0,C 180,E1 -11840.668,E2 -11840.668} C_VEL
LIN {X 0,Y 381.966,Z 519.831,A -85,B 0,C 180,E1 -11842.613,E2 -11842.613} C_VEL
LIN {X 0,Y 382.411,Z 515.002,A -85,B 0,C 180,E1 -11844.647,E2 -11844.647} C_VEL
LIN {X 0,Y 382.904,Z 510.153,A -85,B 0,C 180,E1 -11846.164,E2 -11846.164} C_VEL
LIN {X 0,Y 383.571,Z 503.097,A -85,B 0,C 180,E1 -11847.903,E2 -11847.903} C_VEL
LIN {X 0,Y 384.494,Z 494.607,A -85,B 0,C 180,E1 -11849.555,E2 -11849.555} C_VEL
LIN {X 0,Y 385.274,Z 486.574,A -85,B 0,C 180,E1 -11850.824,E2 -11850.824} C_VEL
LIN {X 0,Y 386.174,Z 476.833,A -85,B 0,C 180,E1 -11852.084,E2 -11852.084} C_VEL
LIN {X 0,Y 387.107,Z 466.563,A -85,B 0,C 180,E1 -11853.152,E2 -11853.152} C_VEL
LIN {X 0,Y 388.047,Z 454.316,A -85,B 0,C 180,E1 -11854.163,E2 -11854.163} C_VEL
LIN {X 0,Y 388.842,Z 442.023,A -85,B 0,C 180,E1 -11854.925,E2 -11854.925} C_VEL
LIN {X 0,Y 389.336,Z 428.996,A -85,B 0,C 180,E1 -11855.508,E2 -11855.508} C_VEL
LIN {X 0,Y 389.812,Z 415.844,A -85,B 0,C 180,E1 -11855.871,E2 -11855.871} C_VEL
LIN {X 0,Y 391.354,Z 336.505,A -85,B 0,C 180,E1 -11857.485,E2 -11857.485} C_VEL
LIN {X 0,Y 387.487,Z 318.732,A -85,B 0,C 180,E1 -11858.137,E2 -11858.137} C_VEL
LIN {X 0,Y 385.567,Z 313.655,A -85,B 0,C 180,E1 -11858.409,E2 -11858.409} C_VEL
LIN {X 0,Y 383.075,Z 302.771,A -85,B 0,C 180,E1 -11860.925,E2 -11860.925} C_VEL
LIN {X 0,Y 383.083,Z 302.771,A -85,B 0,C 180,E1 -11864.026,E2 -11864.026} C_VEL
LIN {X 0,Y 383.139,Z 302.763,A -85,B 0,C 180,E1 -11867.284,E2 -11867.284} C_VEL
LIN {X 0,Y 383.263,Z 302.745,A -85,B 0,C 180,E1 -11871.564,E2 -11871.564} C_VEL
LIN {X 0,Y 383.199,Z 302.752,A -85,B 0,C 180,E1 -11874.738,E2 -11874.738} C_VEL
LIN {X 0,Y 383.387,Z 302.728,A -85,B 0,C 180,E1 -11877.899,E2 -11877.899} C_VEL
LIN {X 0,Y 383.519,Z 302.713,A -85,B 0,C 180,E1 -11880,E2 -11880} C_VEL
LIN {X 0,Y 383.248,Z 302.743,A -85,B 0,C 180,E1 -11883.153,E2 -11883.153} C_VEL
LIN {X 0,Y 383.264,Z 302.74,A -85,B 0,C 180,E1 -11886.316,E2 -11886.316} C_VEL
LIN {X 0,Y 383.152,Z 302.755,A -85,B 0,C 180,E1 -11889.502,E2 -11889.502} C_VEL
LIN {X 0,Y 383.127,Z 302.754,A -85,B 0,C 180,E1 -11893.536,E2 -11893.536} C_VEL
LIN {X 0,Y 383.096,Z 302.758,A -85,B 0,C 180,E1 -11897.069,E2 -11897.069} C_VEL
LIN {X 0,Y 383.03,Z 302.768,A -85,B 0,C 180,E1 -11900.647,E2 -11900.647} C_VEL
LIN {X 0,Y 383.027,Z 302.768,A -85,B 0,C 180,E1 -11903.808,E2 -11903.808} C_VEL
LIN {X 0,Y 383.082,Z 302.763,A -85,B 0,C 180,E1 -11906.123,E2 -11906.123} C_VEL
LIN {X 0,Y 382.994,Z 302.775,A -85,B 0,C 180,E1 -11909.7,E2 -11909.7} C_VEL
LIN {X 0,Y 383.004,Z 302.775,A -85,B 0,C 180,E1 -11913.401,E2 -11913.401} C_VEL
LIN {X 0,Y 383.033,Z 302.771,A -85,B 0,C 180,E1 -11916.164,E2 -11916.164} C_VEL
LIN {X 0,Y 383.01,Z 302.773,A -85,B 0,C 180,E1 -11919.958,E2 -11919.958} C_VEL
LIN {X 0,Y 383.007,Z 302.777,A -85,B 0,C 180,E1 -11922.778,E2 -11922.778} C_VEL
LIN {X 0,Y 382.999,Z 302.776,A -85,B 0,C 180,E1 -11925.789,E2 -11925.789} C_VEL
LIN {X 0,Y 382.99,Z 302.776,A -85,B 0,C 180,E1 -11928.796,E2 -11928.796} C_VEL
LIN {X 0,Y 383,Z 302.78,A -85,B 0,C 180,E1 -11932.096,E2 -11932.096} C_VEL
LIN {X 0,Y 383.02,Z 302.78,A -85,B 0,C 180,E1 -11935.332,E2 -11935.332} C_VEL
LIN {X 0,Y 382.985,Z 302.782,A -85,B 0,C 180,E1 -11939.081,E2 -11939.081} C_VEL
LIN {X 0,Y 383.037,Z 302.831,A -85,B 0,C 180,E1 -11940.719,E2 -11940.719} C_VEL
LIN {X 0,Y 385.733,Z 314.582,A -85,B 0,C 180,E1 -11943.496,E2 -11943.496} C_VEL
LIN {X 0,Y 386.819,Z 321.31,A -85,B 0,C 180,E1 -11945.012,E2 -11945.012} C_VEL
LIN {X 0,Y 385.516,Z 338.946,A -85,B 0,C 180,E1 -11948.616,E2 -11948.616} C_VEL
LIN {X 0,Y 385.485,Z 339.202,A -85,B 0,C 180,E1 -11948.667,E2 -11948.667} C_VEL
LIN {X 0,Y 389.367,Z 361.031,A -85,B 0,C 180,E1 -11949.408,E2 -11949.408} C_VEL
LIN {X 0,Y 390.887,Z 372.346,A -85,B 0,C 180,E1 -11949.75,E2 -11949.75} C_VEL
LIN {X 0,Y 389.373,Z 448.719,A -85,B 0,C 180,E1 -11951.314,E2 -11951.314} C_VEL
LIN {X 0,Y 388.673,Z 462.277,A -85,B 0,C 180,E1 -11951.791,E2 -11951.791} C_VEL
LIN {X 0,Y 387.845,Z 475.191,A -85,B 0,C 180,E1 -11952.466,E2 -11952.466} C_VEL
LIN {X 0,Y 386.96,Z 486.207,A -85,B 0,C 180,E1 -11953.242,E2 -11953.242} C_VEL
LIN {X 0,Y 385.92,Z 497.77,A -85,B 0,C 180,E1 -11954.282,E2 -11954.282} C_VEL
LIN {X 0,Y 384.955,Z 508.486,A -85,B 0,C 180,E1 -11955.493,E2 -11955.493} C_VEL
LIN {X 0,Y 384.107,Z 517.667,A -85,B 0,C 180,E1 -11956.778,E2 -11956.778} C_VEL
LIN {X 0,Y 383.123,Z 526.827,A -85,B 0,C 180,E1 -11958.358,E2 -11958.358} C_VEL
LIN {X 0,Y 382.465,Z 534.234,A -85,B 0,C 180,E1 -11959.946,E2 -11959.946} C_VEL
LIN {X 0,Y 382.056,Z 540.176,A -85,B 0,C 180,E1 -11961.537,E2 -11961.537} C_VEL
LIN {X 0,Y 381.78,Z 544.86,A -85,B 0,C 180,E1 -11963.127,E2 -11963.127} C_VEL
LIN {X 0,Y 381.64,Z 548.431,A -85,B 0,C 180,E1 -11964.716,E2 -11964.716} C_VEL
LIN {X 0,Y 381.626,Z 550.223,A -85,B 0,C 180,E1 -11965.775,E2 -11965.775} C_VEL
LIN {X 0,Y 381.599,Z 552.566,A -85,B 0,C 180,E1 -11967.888,E2 -11967.888} C_VEL
LIN {X 0,Y 381.652,Z 553.123,A -85,B 0,C 180,E1 -11968.944,E2 -11968.944} C_VEL
LIN {X 0,Y 381.657,Z 553.235,A -85,B 0,C 180,E1 -11969.999,E2 -11969.999} C_VEL
LIN {X 0,Y 381.67,Z 552.95,A -85,B 0,C 180,E1 -11971.054,E2 -11971.054} C_VEL
LIN {X 0,Y 381.602,Z 552.265,A -85,B 0,C 180,E1 -11972.11,E2 -11972.11} C_VEL
LIN {X 0,Y 381.553,Z 551.155,A -85,B 0,C 180,E1 -11973.167,E2 -11973.167} C_VEL
LIN {X 0,Y 381.629,Z 549.591,A -85,B 0,C 180,E1 -11974.224,E2 -11974.224} C_VEL
LIN {X 0,Y 381.686,Z 545.694,A -85,B 0,C 180,E1 -11976.118,E2 -11976.118} C_VEL
LIN {X 0,Y 381.916,Z 540.503,A -85,B 0,C 180,E1 -11977.932,E2 -11977.932} C_VEL
LIN {X 0,Y 382.36,Z 533.442,A -85,B 0,C 180,E1 -11979.788,E2 -11979.788} C_VEL
LIN {X 0,Y 382.907,Z 525.784,A -85,B 0,C 180,E1 -11981.379,E2 -11981.379} C_VEL
LIN {X 0,Y 383.598,Z 517.956,A -85,B 0,C 180,E1 -11982.7,E2 -11982.7} C_VEL
LIN {X 0,Y 384.364,Z 508.644,A -85,B 0,C 180,E1 -11983.987,E2 -11983.987} C_VEL
LIN {X 0,Y 385.173,Z 497.745,A -85,B 0,C 180,E1 -11985.205,E2 -11985.205} C_VEL
LIN {X 0,Y 386.063,Z 485.908,A -85,B 0,C 180,E1 -11986.253,E2 -11986.253} C_VEL
LIN {X 0,Y 386.931,Z 473.272,A -85,B 0,C 180,E1 -11987.098,E2 -11987.098} C_VEL
LIN {X 0,Y 387.674,Z 460.005,A -85,B 0,C 180,E1 -11987.745,E2 -11987.745} C_VEL
LIN {X 0,Y 388.186,Z 446.487,A -85,B 0,C 180,E1 -11988.163,E2 -11988.163} C_VEL
LIN {X 0,Y 389.338,Z 370.939,A -85,B 0,C 180,E1 -11989.67,E2 -11989.67} C_VEL
LIN {X 0,Y 384.936,Z 341.069,A -85,B 0,C 180,E1 -11990.506,E2 -11990.506} C_VEL
LIN {X 0,Y 386.309,Z 324.049,A -85,B 0,C 180,E1 -11994.132,E2 -11994.132} C_VEL
LIN {X 0,Y 386.489,Z 320.015,A -85,B 0,C 180,E1 -11995.01,E2 -11995.01} C_VEL
LIN {X 0,Y 384.484,Z 309.424,A -85,B 0,C 180,E1 -11997.486,E2 -11997.486} C_VEL
LIN {X 0,Y 383.06,Z 302.769,A -85,B 0,C 180,E1 -11999.127,E2 -11999.127} C_VEL
LIN {X 0,Y 382.985,Z 302.783,A -85,B 0,C 180,E1 -12002.421,E2 -12002.421} C_VEL
LIN {X 0,Y 383.022,Z 302.773,A -85,B 0,C 180,E1 -12005.955,E2 -12005.955} C_VEL
LIN {X 0,Y 383.01,Z 302.772,A -85,B 0,C 180,E1 -12009.585,E2 -12009.585} C_VEL
LIN {X 0,Y 383.001,Z 302.776,A -85,B 0,C 180,E1 -12012.778,E2 -12012.778} C_VEL
LIN {X 0,Y 382.995,Z 302.774,A -85,B 0,C 180,E1 -12015.789,E2 -12015.789} C_VEL
LIN {X 0,Y 382.986,Z 302.779,A -85,B 0,C 180,E1 -12018.795,E2 -12018.795} C_VEL
LIN {X 0,Y 382.997,Z 302.774,A -85,B 0,C 180,E1 -12022.095,E2 -12022.095} C_VEL
LIN {X 0,Y 383.013,Z 302.772,A -85,B 0,C 180,E1 -12025.332,E2 -12025.332} C_VEL
LIN {X 0,Y 382.978,Z 302.78,A -85,B 0,C 180,E1 -12029.081,E2 -12029.081} C_VEL
LIN {X 0,Y 383.051,Z 302.77,A -85,B 0,C 180,E1 -12032.698,E2 -12032.698} C_VEL
LIN {X 0,Y 383.047,Z 302.774,A -85,B 0,C 180,E1 -12035.039,E2 -12035.039} C_VEL
LIN {X 0,Y 382.987,Z 302.775,A -85,B 0,C 180,E1 -12038.469,E2 -12038.469} C_VEL
LIN {X 0,Y 383.083,Z 302.763,A -85,B 0,C 180,E1 -12041.828,E2 -12041.828} C_VEL
LIN {X 0,Y 383.104,Z 302.764,A -85,B 0,C 180,E1 -12045.118,E2 -12045.118} C_VEL
LIN {X 0,Y 383.091,Z 302.761,A -85,B 0,C 180,E1 -12048.358,E2 -12048.358} C_VEL
LIN {X 0,Y 383.298,Z 302.738,A -85,B 0,C 180,E1 -12051.933,E2 -12051.933} C_VEL
LIN {X 0,Y 383.193,Z 302.749,A -85,B 0,C 180,E1 -12054.739,E2 -12054.739} C_VEL
LIN {X 0,Y 383.379,Z 302.73,A -85,B 0,C 180,E1 -12057.899,E2 -12057.899} C_VEL
LIN {X 0,Y 383.511,Z 302.713,A -85,B 0,C 180,E1 -12060,E2 -12060} C_VEL
LIN {X 0,Y 383.242,Z 302.743,A -85,B 0,C 180,E1 -12063.154,E2 -12063.154} C_VEL
LIN {X 0,Y 383.241,Z 302.744,A -85,B 0,C 180,E1 -12066.482,E2 -12066.482} C_VEL
LIN {X 0,Y 383.145,Z 302.756,A -85,B 0,C 180,E1 -12069.503,E2 -12069.503} C_VEL
LIN {X 0,Y 383.12,Z 302.759,A -85,B 0,C 180,E1 -12073.537,E2 -12073.537} C_VEL
LIN {X 0,Y 383.089,Z 302.762,A -85,B 0,C 180,E1 -12077.455,E2 -12077.455} C_VEL
LIN {X 0,Y 383.024,Z 302.773,A -85,B 0,C 180,E1 -12080.647,E2 -12080.647} C_VEL
LIN {X 0,Y 383.012,Z 302.772,A -85,B 0,C 180,E1 -12083.809,E2 -12083.809} C_VEL
LIN {X 0,Y 382.989,Z 302.774,A -85,B 0,C 180,E1 -12087.308,E2 -12087.308} C_VEL
LIN {X 0,Y 382.978,Z 302.778,A -85,B 0,C 180,E1 -12090.92,E2 -12090.92} C_VEL
LIN {X 0,Y 383.015,Z 302.778,A -85,B 0,C 180,E1 -12094.669,E2 -12094.669} C_VEL
LIN {X 0,Y 382.993,Z 302.773,A -85,B 0,C 180,E1 -12097.904,E2 -12097.904} C_VEL
LIN {X 0,Y 382.977,Z 302.777,A -85,B 0,C 180,E1 -12101.349,E2 -12101.349} C_VEL
LIN {X 0,Y 382.993,Z 302.774,A -85,B 0,C 180,E1 -12104.304,E2 -12104.304} C_VEL
LIN {X 0,Y 383.009,Z 302.776,A -85,B 0,C 180,E1 -12107.241,E2 -12107.241} C_VEL
LIN {X 0,Y 382.985,Z 302.775,A -85,B 0,C 180,E1 -12110.42,E2 -12110.42} C_VEL
LIN {X 0,Y 383.024,Z 302.77,A -85,B 0,C 180,E1 -12114.045,E2 -12114.045} C_VEL
LIN {X 0,Y 382.986,Z 302.778,A -85,B 0,C 180,E1 -12117.579,E2 -12117.579} C_VEL
LIN {X 0,Y 382.977,Z 302.775,A -85,B 0,C 180,E1 -12120.3,E2 -12120.3} C_VEL
LIN {X 0,Y 383.003,Z 302.773,A -85,B 0,C 180,E1 -12124.046,E2 -12124.046} C_VEL
LIN {X 0,Y 382.991,Z 302.778,A -85,B 0,C 180,E1 -12127.335,E2 -12127.335} C_VEL
LIN {X 0,Y 383.061,Z 302.765,A -85,B 0,C 180,E1 -12130.717,E2 -12130.717} C_VEL
LIN {X 0,Y 383.082,Z 302.766,A -85,B 0,C 180,E1 -12134.027,E2 -12134.027} C_VEL
LIN {X 0,Y 383.137,Z 302.757,A -85,B 0,C 180,E1 -12137.285,E2 -12137.285} C_VEL
LIN {X 0,Y 383.139,Z 302.756,A -85,B 0,C 180,E1 -12140.498,E2 -12140.498} C_VEL
LIN {X 0,Y 383.237,Z 302.746,A -85,B 0,C 180,E1 -12143.684,E2 -12143.684} C_VEL
LIN {X 0,Y 383.368,Z 302.731,A -85,B 0,C 180,E1 -12147.899,E2 -12147.899} C_VEL
LIN {X 0,Y 383.263,Z 302.74,A -85,B 0,C 180,E1 -12151.051,E2 -12151.051} C_VEL
LIN {X 0,Y 383.367,Z 302.733,A -85,B 0,C 180,E1 -12152.102,E2 -12152.102} C_VEL
LIN {X 0,Y 383.237,Z 302.75,A -85,B 0,C 180,E1 -12156.318,E2 -12156.318} C_VEL
LIN {X 0,Y 383.178,Z 302.757,A -85,B 0,C 180,E1 -12158.438,E2 -12158.438} C_VEL
LIN {X 0,Y 383.082,Z 302.762,A -85,B 0,C 180,E1 -12161.643,E2 -12161.643} C_VEL
LIN {X 0,Y 383.057,Z 302.766,A -85,B 0,C 180,E1 -12163.799,E2 -12163.799} C_VEL
LIN {X 0,Y 383.057,Z 302.766,A -85,B 0,C 180,E1 -12167.434,E2 -12167.434} C_VEL
LIN {X 0,Y 383.019,Z 302.776,A -85,B 0,C 180,E1 -12170.641,E2 -12170.641} C_VEL
LIN {X 0,Y 383.094,Z 302.942,A -85,B 0,C 180,E1 -12173.684,E2 -12173.684} C_VEL
LIN {X 0,Y 385.129,Z 313.898,A -85,B 0,C 180,E1 -12176.577,E2 -12176.577} C_VEL
LIN {X 0,Y 389.703,Z 336.502,A -85,B 0,C 180,E1 -12177.278,E2 -12177.278} C_VEL
LIN {X 0,Y 389.606,Z 348.731,A -85,B 0,C 180,E1 -12177.525,E2 -12177.525} C_VEL
LIN {X 0,Y 388.898,Z 354.565,A -85,B 0,C 180,E1 -12177.612,E2 -12177.612} C_VEL
LIN {X 0,Y 383.03,Z 373.512,A -85,B 0,C 180,E1 -12177.738,E2 -12177.738} C_VEL
LIN {X 0,Y 382.231,Z 379.35,A -85,B 0,C 180,E1 -12177.823,E2 -12177.823} C_VEL
LIN {X 0,Y 381.44,Z 422.373,A -85,B 0,C 180,E1 -12178.718,E2 -12178.718} C_VEL
LIN {X 0,Y 380.873,Z 436.336,A -85,B 0,C 180,E1 -12179.237,E2 -12179.237} C_VEL
LIN {X 0,Y 380.343,Z 448.77,A -85,B 0,C 180,E1 -12179.928,E2 -12179.928} C_VEL
LIN {X 0,Y 379.561,Z 460.157,A -85,B 0,C 180,E1 -12180.765,E2 -12180.765} C_VEL
LIN {X 0,Y 378.708,Z 471.406,A -85,B 0,C 180,E1 -12181.819,E2 -12181.819} C_VEL
LIN {X 0,Y 377.928,Z 482.113,A -85,B 0,C 180,E1 -12183.085,E2 -12183.085} C_VEL
LIN {X 0,Y 377.097,Z 491.474,A -85,B 0,C 180,E1 -12184.458,E2 -12184.458} C_VEL
LIN {X 0,Y 376.319,Z 499.692,A -85,B 0,C 180,E1 -12185.937,E2 -12185.937} C_VEL
LIN {X 0,Y 375.72,Z 506.488,A -85,B 0,C 180,E1 -12187.44,E2 -12187.44} C_VEL
LIN {X 0,Y 375.234,Z 512.83,A -85,B 0,C 180,E1 -12189.207,E2 -12189.207} C_VEL
LIN {X 0,Y 374.888,Z 517.768,A -85,B 0,C 180,E1 -12191.007,E2 -12191.007} C_VEL
LIN {X 0,Y 374.571,Z 521.649,A -85,B 0,C 180,E1 -12192.966,E2 -12192.966} C_VEL
LIN {X 0,Y 374.393,Z 523.636,A -85,B 0,C 180,E1 -12194.493,E2 -12194.493} C_VEL
LIN {X 0,Y 374.349,Z 524.784,A -85,B 0,C 180,E1 -12196.001,E2 -12196.001} C_VEL
LIN {X 0,Y 374.36,Z 525.152,A -85,B 0,C 180,E1 -12197.48,E2 -12197.48} C_VEL
LIN {X 0,Y 374.383,Z 524.759,A -85,B 0,C 180,E1 -12198.926,E2 -12198.926} C_VEL
LIN {X 0,Y 374.479,Z 523.639,A -85,B 0,C 180,E1 -12200.35,E2 -12200.35} C_VEL
LIN {X 0,Y 374.747,Z 521.498,A -85,B 0,C 180,E1 -12201.968,E2 -12201.968} C_VEL
LIN {X 0,Y 375.071,Z 518.164,A -85,B 0,C 180,E1 -12203.681,E2 -12203.681} C_VEL
LIN {X 0,Y 375.578,Z 513.537,A -85,B 0,C 180,E1 -12205.422,E2 -12205.422} C_VEL
LIN {X 0,Y 376.247,Z 507.378,A -85,B 0,C 180,E1 -12207.2,E2 -12207.2} C_VEL
LIN {X 0,Y 376.978,Z 500.244,A -85,B 0,C 180,E1 -12208.816,E2 -12208.816} C_VEL
LIN {X 0,Y 377.978,Z 491.542,A -85,B 0,C 180,E1 -12210.393,E2 -12210.393} C_VEL
LIN {X 0,Y 378.896,Z 482.177,A -85,B 0,C 180,E1 -12211.771,E2 -12211.771} C_VEL
LIN {X 0,Y 379.981,Z 471.15,A -85,B 0,C 180,E1 -12213.058,E2 -12213.058} C_VEL
LIN {X 0,Y 380.926,Z 460.108,A -85,B 0,C 180,E1 -12214.085,E2 -12214.085} C_VEL
LIN {X 0,Y 381.791,Z 449.518,A -85,B 0,C 180,E1 -12214.858,E2 -12214.858} C_VEL
LIN {X 0,Y 382.439,Z 436.597,A -85,B 0,C 180,E1 -12215.576,E2 -12215.576} C_VEL
LIN {X 0,Y 382.982,Z 424.21,A -85,B 0,C 180,E1 -12216.045,E2 -12216.045} C_VEL
LIN {X 0,Y 383.601,Z 396.693,A -85,B 0,C 180,E1 -12216.654,E2 -12216.654} C_VEL
LIN {X 0,Y 384.922,Z 337.97,A -85,B 0,C 180,E1 -12217.878,E2 -12217.878} C_VEL
LIN {X 0,Y 381.37,Z 321.414,A -85,B 0,C 180,E1 -12218.496,E2 -12218.496} C_VEL
LIN {X 0,Y 378.422,Z 313.945,A -85,B 0,C 180,E1 -12218.91,E2 -12218.91} C_VEL
LIN {X 0,Y 376.03,Z 303.65,A -85,B 0,C 180,E1 -12221.368,E2 -12221.368} C_VEL
LIN {X 0,Y 376.061,Z 303.647,A -85,B 0,C 180,E1 -12224.832,E2 -12224.832} C_VEL
LIN {X 0,Y 376.051,Z 303.642,A -85,B 0,C 180,E1 -12228.136,E2 -12228.136} C_VEL
LIN {X 0,Y 376.26,Z 303.617,A -85,B 0,C 180,E1 -12231.878,E2 -12231.878} C_VEL
LIN {X 0,Y 376.171,Z 303.627,A -85,B 0,C 180,E1 -12234.64,E2 -12234.64} C_VEL
LIN {X 0,Y 376.353,Z 303.605,A -85,B 0,C 180,E1 -12237.859,E2 -12237.859} C_VEL
LIN {X 0,Y 376.489,Z 303.588,A -85,B 0,C 180,E1 -12240,E2 -12240} C_VEL
LIN {X 0,Y 376.186,Z 303.623,A -85,B 0,C 180,E1 -12243.213,E2 -12243.213} C_VEL
LIN {X 0,Y 376.221,Z 303.616,A -85,B 0,C 180,E1 -12246.435,E2 -12246.435} C_VEL
LIN {X 0,Y 376.12,Z 303.632,A -85,B 0,C 180,E1 -12249.681,E2 -12249.681} C_VEL
LIN {X 0,Y 376.091,Z 303.63,A -85,B 0,C 180,E1 -12253.657,E2 -12253.657} C_VEL
LIN {X 0,Y 376.034,Z 303.637,A -85,B 0,C 180,E1 -12257.4,E2 -12257.4} C_VEL
LIN {X 0,Y 375.98,Z 303.646,A -85,B 0,C 180,E1 -12260.832,E2 -12260.832} C_VEL
LIN {X 0,Y 375.991,Z 303.645,A -85,B 0,C 180,E1 -12264.282,E2 -12264.282} C_VEL
LIN {X 0,Y 376.022,Z 303.647,A -85,B 0,C 180,E1 -12266.652,E2 -12266.652} C_VEL
LIN {X 0,Y 375.966,Z 303.651,A -85,B 0,C 180,E1 -12270.312,E2 -12270.312} C_VEL
LIN {X 0,Y 375.961,Z 303.65,A -85,B 0,C 180,E1 -12274.111,E2 -12274.111} C_VEL
LIN {X 0,Y 375.955,Z 303.655,A -85,B 0,C 180,E1 -12276.741,E2 -12276.741} C_VEL
LIN {X 0,Y 375.99,Z 303.648,A -85,B 0,C 180,E1 -12279.97,E2 -12279.97} C_VEL
LIN {X 0,Y 375.931,Z 303.657,A -85,B 0,C 180,E1 -12283.766,E2 -12283.766} C_VEL
LIN {X 0,Y 375.935,Z 303.656,A -85,B 0,C 180,E1 -12286.81,E2 -12286.81} C_VEL
LIN {X 0,Y 375.963,Z 303.653,A -85,B 0,C 180,E1 -12290.537,E2 -12290.537} C_VEL
LIN {X 0,Y 375.966,Z 303.657,A -85,B 0,C 180,E1 -12293.495,E2 -12293.495} C_VEL
LIN {X 0,Y 375.962,Z 303.661,A -85,B 0,C 180,E1 -12295.888,E2 -12295.888} C_VEL
LIN {X 0,Y 375.968,Z 303.654,A -85,B 0,C 180,E1 -12299.687,E2 -12299.687} C_VEL
LIN {X 0,Y 375.999,Z 303.742,A -85,B 0,C 180,E1 -12300.308,E2 -12300.308} C_VEL
LIN {X 0,Y 378.582,Z 314.859,A -85,B 0,C 180,E1 -12303.008,E2 -12303.008} C_VEL
LIN {X 0,Y 379.946,Z 322.717,A -85,B 0,C 180,E1 -12304.821,E2 -12304.821} C_VEL
LIN {X 0,Y 378.697,Z 338.887,A -85,B 0,C 180,E1 -12308.195,E2 -12308.195} C_VEL
LIN {X 0,Y 382.595,Z 360.055,A -85,B 0,C 180,E1 -12308.945,E2 -12308.945} C_VEL
LIN {X 0,Y 384.354,Z 373.271,A -85,B 0,C 180,E1 -12309.358,E2 -12309.358} C_VEL
LIN {X 0,Y 382.728,Z 448.687,A -85,B 0,C 180,E1 -12310.942,E2 -12310.942} C_VEL
LIN {X 0,Y 381.998,Z 462.148,A -85,B 0,C 180,E1 -12311.426,E2 -12311.426} C_VEL
LIN {X 0,Y 381.153,Z 474.485,A -85,B 0,C 180,E1 -12312.079,E2 -12312.079} C_VEL
LIN {X 0,Y 380.191,Z 486.396,A -85,B 0,C 180,E1 -12312.934,E2 -12312.934} C_VEL
LIN {X 0,Y 379.073,Z 497.879,A -85,B 0,C 180,E1 -12313.991,E2 -12313.991} C_VEL
LIN {X 0,Y 378.183,Z 507.483,A -85,B 0,C 180,E1 -12315.094,E2 -12315.094} C_VEL
LIN {X 0,Y 377.334,Z 515.905,A -85,B 0,C 180,E1 -12316.262,E2 -12316.262} C_VEL
LIN {X 0,Y 376.503,Z 523.95,A -85,B 0,C 180,E1 -12317.604,E2 -12317.604} C_VEL
LIN {X 0,Y 375.646,Z 531.835,A -85,B 0,C 180,E1 -12319.216,E2 -12319.216} C_VEL
LIN {X 0,Y 375.162,Z 538.17,A -85,B 0,C 180,E1 -12320.837,E2 -12320.837} C_VEL
LIN {X 0,Y 374.795,Z 543.22,A -85,B 0,C 180,E1 -12322.457,E2 -12322.457} C_VEL
LIN {X 0,Y 374.582,Z 546.841,A -85,B 0,C 180,E1 -12323.934,E2 -12323.934} C_VEL
LIN {X 0,Y 374.551,Z 550.002,A -85,B 0,C 180,E1 -12325.695,E2 -12325.695} C_VEL
LIN {X 0,Y 374.497,Z 552.326,A -85,B 0,C 180,E1 -12327.848,E2 -12327.848} C_VEL
LIN {X 0,Y 374.567,Z 552.862,A -85,B 0,C 180,E1 -12328.924,E2 -12328.924} C_VEL
LIN {X 0,Y 374.59,Z 552.963,A -85,B 0,C 180,E1 -12329.999,E2 -12329.999} C_VEL
LIN {X 0,Y 374.583,Z 552.666,A -85,B 0,C 180,E1 -12331.074,E2 -12331.074} C_VEL
LIN {X 0,Y 374.502,Z 551.968,A -85,B 0,C 180,E1 -12332.15,E2 -12332.15} C_VEL
LIN {X 0,Y 374.467,Z 550.832,A -85,B 0,C 180,E1 -12333.227,E2 -12333.227} C_VEL
LIN {X 0,Y 374.542,Z 548.326,A -85,B 0,C 180,E1 -12334.843,E2 -12334.843} C_VEL
LIN {X 0,Y 374.63,Z 544.774,A -85,B 0,C 180,E1 -12336.462,E2 -12336.462} C_VEL
LIN {X 0,Y 374.859,Z 540.086,A -85,B 0,C 180,E1 -12338.083,E2 -12338.083} C_VEL
LIN {X 0,Y 375.23,Z 534.117,A -85,B 0,C 180,E1 -12339.704,E2 -12339.704} C_VEL
LIN {X 0,Y 375.777,Z 526.656,A -85,B 0,C 180,E1 -12341.324,E2 -12341.324} C_VEL
LIN {X 0,Y 376.604,Z 517.381,A -85,B 0,C 180,E1 -12342.94,E2 -12342.94} C_VEL
LIN {X 0,Y 377.51,Z 507.113,A -85,B 0,C 180,E1 -12344.358,E2 -12344.358} C_VEL
LIN {X 0,Y 378.347,Z 495.692,A -85,B 0,C 180,E1 -12345.625,E2 -12345.625} C_VEL
LIN {X 0,Y 379.339,Z 483.233,A -85,B 0,C 180,E1 -12346.688,E2 -12346.688} C_VEL
LIN {X 0,Y 380.21,Z 471.072,A -85,B 0,C 180,E1 -12347.479,E2 -12347.479} C_VEL
LIN {X 0,Y 380.923,Z 458.492,A -85,B 0,C 180,E1 -12348.07,E2 -12348.07} C_VEL
LIN {X 0,Y 381.379,Z 445.605,A -85,B 0,C 180,E1 -12348.464,E2 -12348.464} C_VEL
LIN {X 0,Y 382.517,Z 371.652,A -85,B 0,C 180,E1 -12349.97,E2 -12349.97} C_VEL
LIN {X 0,Y 378.047,Z 340.797,A -85,B 0,C 180,E1 -12350.856,E2 -12350.856} C_VEL
LIN {X 0,Y 379.443,Z 324.189,A -85,B 0,C 180,E1 -12354.466,E2 -12354.466} C_VEL
LIN {X 0,Y 379.473,Z 320.851,A -85,B 0,C 180,E1 -12355.211,E2 -12355.211} C_VEL
LIN {X 0,Y 376.932,Z 307.963,A -85,B 0,C 180,E1 -12358.303,E2 -12358.303} C_VEL
LIN {X 0,Y 375.991,Z 303.651,A -85,B 0,C 180,E1 -12359.383,E2 -12359.383} C_VEL
LIN {X 0,Y 375.949,Z 303.656,A -85,B 0,C 180,E1 -12362.828,E2 -12362.828} C_VEL
LIN {X 0,Y 375.955,Z 303.65,A -85,B 0,C 180,E1 -12365.415,E2 -12365.415} C_VEL
LIN {X 0,Y 375.969,Z 303.655,A -85,B 0,C 180,E1 -12368.269,E2 -12368.269} C_VEL
LIN {X 0,Y 375.931,Z 303.653,A -85,B 0,C 180,E1 -12371.6,E2 -12371.6} C_VEL
LIN {X 0,Y 375.925,Z 303.654,A -85,B 0,C 180,E1 -12375.268,E2 -12375.268} C_VEL
LIN {X 0,Y 375.932,Z 303.658,A -85,B 0,C 180,E1 -12378.398,E2 -12378.398} C_VEL
LIN {X 0,Y 375.972,Z 303.648,A -85,B 0,C 180,E1 -12381.729,E2 -12381.729} C_VEL
LIN {X 0,Y 375.975,Z 303.649,A -85,B 0,C 180,E1 -12385.332,E2 -12385.332} C_VEL
LIN {X 0,Y 375.953,Z 303.653,A -85,B 0,C 180,E1 -12388.438,E2 -12388.438} C_VEL
LIN {X 0,Y 375.978,Z 303.647,A -85,B 0,C 180,E1 -12392.14,E2 -12392.14} C_VEL
LIN {X 0,Y 376.001,Z 303.646,A -85,B 0,C 180,E1 -12394.539,E2 -12394.539} C_VEL
LIN {X 0,Y 375.957,Z 303.65,A -85,B 0,C 180,E1 -12398.046,E2 -12398.046} C_VEL
LIN {X 0,Y 376.018,Z 303.646,A -85,B 0,C 180,E1 -12401.474,E2 -12401.474} C_VEL
LIN {X 0,Y 376.053,Z 303.64,A -85,B 0,C 180,E1 -12404.833,E2 -12404.833} C_VEL
LIN {X 0,Y 376.044,Z 303.64,A -85,B 0,C 180,E1 -12408.137,E2 -12408.137} C_VEL
LIN {X 0,Y 376.252,Z 303.616,A -85,B 0,C 180,E1 -12411.877,E2 -12411.877} C_VEL
LIN {X 0,Y 376.165,Z 303.624,A -85,B 0,C 180,E1 -12414.64,E2 -12414.64} C_VEL
LIN {X 0,Y 376.345,Z 303.606,A -85,B 0,C 180,E1 -12417.86,E2 -12417.86} C_VEL
LIN {X 0,Y 376.481,Z 303.588,A -85,B 0,C 180,E1 -12420,E2 -12420} C_VEL
LIN {X 0,Y 376.18,Z 303.623,A -85,B 0,C 180,E1 -12423.213,E2 -12423.213} C_VEL
LIN {X 0,Y 376.21,Z 303.62,A -85,B 0,C 180,E1 -12426.466,E2 -12426.466} C_VEL
LIN {X 0,Y 376.113,Z 303.634,A -85,B 0,C 180,E1 -12429.682,E2 -12429.682} C_VEL
LIN {X 0,Y 376.084,Z 303.636,A -85,B 0,C 180,E1 -12433.658,E2 -12433.658} C_VEL
LIN {X 0,Y 376.039,Z 303.641,A -85,B 0,C 180,E1 -12437.608,E2 -12437.608} C_VEL
LIN {X 0,Y 375.974,Z 303.649,A -85,B 0,C 180,E1 -12440.833,E2 -12440.833} C_VEL
LIN {X 0,Y 375.973,Z 303.654,A -85,B 0,C 180,E1 -12444.283,E2 -12444.283} C_VEL
LIN {X 0,Y 375.931,Z 303.654,A -85,B 0,C 180,E1 -12447.864,E2 -12447.864} C_VEL
LIN {X 0,Y 375.953,Z 303.65,A -85,B 0,C 180,E1 -12451.563,E2 -12451.563} C_VEL
LIN {X 0,Y 375.954,Z 303.651,A -85,B 0,C 180,E1 -12455.416,E2 -12455.416} C_VEL
LIN {X 0,Y 375.937,Z 303.654,A -85,B 0,C 180,E1 -12458.265,E2 -12458.265} C_VEL
LIN {X 0,Y 375.933,Z 303.66,A -85,B 0,C 180,E1 -12460.869,E2 -12460.869} C_VEL
LIN {X 0,Y 375.927,Z 303.654,A -85,B 0,C 180,E1 -12463.767,E2 -12463.767} C_VEL
LIN {X 0,Y 375.932,Z 303.658,A -85,B 0,C 180,E1 -12466.812,E2 -12466.812} C_VEL
LIN {X 0,Y 375.935,Z 303.654,A -85,B 0,C 180,E1 -12470.535,E2 -12470.535} C_VEL
LIN {X 0,Y 375.962,Z 303.653,A -85,B 0,C 180,E1 -12473.497,E2 -12473.497} C_VEL
LIN {X 0,Y 375.96,Z 303.65,A -85,B 0,C 180,E1 -12475.89,E2 -12475.89} C_VEL
LIN {X 0,Y 375.962,Z 303.652,A -85,B 0,C 180,E1 -12479.688,E2 -12479.688} C_VEL
LIN {X 0,Y 375.918,Z 303.655,A -85,B 0,C 180,E1 -12482.136,E2 -12482.136} C_VEL
LIN {X 0,Y 375.96,Z 303.654,A -85,B 0,C 180,E1 -12485.717,E2 -12485.717} C_VEL
LIN {X 0,Y 376,Z 303.647,A -85,B 0,C 180,E1 -12489.199,E2 -12489.199} C_VEL
LIN {X 0,Y 376.035,Z 303.64,A -85,B 0,C 180,E1 -12492.601,E2 -12492.601} C_VEL
LIN {X 0,Y 376.093,Z 303.634,A -85,B 0,C 180,E1 -12496.343,E2 -12496.343} C_VEL
LIN {X 0,Y 376.11,Z 303.633,A -85,B 0,C 180,E1 -12500.319,E2 -12500.319} C_VEL
LIN {X 0,Y 376.197,Z 303.622,A -85,B 0,C 180,E1 -12503.565,E2 -12503.565} C_VEL
LIN {X 0,Y 376.332,Z 303.607,A -85,B 0,C 180,E1 -12507.86,E2 -12507.86} C_VEL
LIN {X 0,Y 376.234,Z 303.615,A -85,B 0,C 180,E1 -12511.071,E2 -12511.071} C_VEL
LIN {X 0,Y 376.331,Z 303.609,A -85,B 0,C 180,E1 -12512.141,E2 -12512.141} C_VEL
LIN {X 0,Y 376.197,Z 303.626,A -85,B 0,C 180,E1 -12516.436,E2 -12516.436} C_VEL
LIN {X 0,Y 376.139,Z 303.632,A -85,B 0,C 180,E1 -12518.597,E2 -12518.597} C_VEL
LIN {X 0,Y 376.033,Z 303.641,A -85,B 0,C 180,E1 -12521.865,E2 -12521.865} C_VEL
LIN {X 0,Y 376.012,Z 303.645,A -85,B 0,C 180,E1 -12524.063,E2 -12524.063} C_VEL
LIN {X 0,Y 376.011,Z 303.643,A -85,B 0,C 180,E1 -12527.589,E2 -12527.589} C_VEL
LIN {X 0,Y 375.984,Z 303.653,A -85,B 0,C 180,E1 -12530.832,E2 -12530.832} C_VEL
LIN {X 0,Y 376.03,Z 303.816,A -85,B 0,C 180,E1 -12533.44,E2 -12533.44} C_VEL
LIN {X 0,Y 377.957,Z 314.121,A -85,B 0,C 180,E1 -12536.208,E2 -12536.208} C_VEL
LIN {X 0,Y 379.859,Z 321.375,A -85,B 0,C 180,E1 -12536.475,E2 -12536.475} C_VEL
LIN {X 0,Y 382.968,Z 337.531,A -85,B 0,C 180,E1 -12536.975,E2 -12536.975} C_VEL
LIN {X 0,Y 382.231,Z 379.35,A -85,B 0,C 180,E1 -12537.823,E2 -12537.823} C_VEL
LIN {X 0,Y 381.432,Z 385.187,A -85,B 0,C 180,E1 -12537.908,E2 -12537.908} C_VEL
LIN {X 0,Y 375.588,Z 404.132,A -85,B 0,C 180,E1 -12538.043,E2 -12538.043} C_VEL
LIN {X 0,Y 374.9,Z 409.964,A -85,B 0,C 180,E1 -12538.135,E2 -12538.135} C_VEL
LIN {X 0,Y 374.5,Z 426.353,A -85,B 0,C 180,E1 -12538.542,E2 -12538.542} C_VEL
LIN {X 0,Y 374.006,Z 438.387,A -85,B 0,C 180,E1 -12539.046,E2 -12539.046} C_VEL
LIN {X 0,Y 373.314,Z 451.084,A -85,B 0,C 180,E1 -12539.798,E2 -12539.798} C_VEL
LIN {X 0,Y 372.57,Z 461.676,A -85,B 0,C 180,E1 -12540.619,E2 -12540.619} C_VEL
LIN {X 0,Y 371.701,Z 472.722,A -85,B 0,C 180,E1 -12541.695,E2 -12541.695} C_VEL
LIN {X 0,Y 370.89,Z 483.371,A -85,B 0,C 180,E1 -12543.01,E2 -12543.01} C_VEL
LIN {X 0,Y 370.027,Z 492.555,A -85,B 0,C 180,E1 -12544.406,E2 -12544.406} C_VEL
LIN {X 0,Y 369.242,Z 500.569,A -85,B 0,C 180,E1 -12545.897,E2 -12545.897} C_VEL
LIN {X 0,Y 368.579,Z 507.899,A -85,B 0,C 180,E1 -12547.602,E2 -12547.602} C_VEL
LIN {X 0,Y 368.179,Z 512.913,A -85,B 0,C 180,E1 -12549.045,E2 -12549.045} C_VEL
LIN {X 0,Y 367.905,Z 517.01,A -85,B 0,C 180,E1 -12550.504,E2 -12550.504} C_VEL
LIN {X 0,Y 367.679,Z 520.264,A -85,B 0,C 180,E1 -12551.991,E2 -12551.991} C_VEL
LIN {X 0,Y 367.394,Z 522.758,A -85,B 0,C 180,E1 -12553.524,E2 -12553.524} C_VEL
LIN {X 0,Y 367.293,Z 524.432,A -85,B 0,C 180,E1 -12555.071,E2 -12555.071} C_VEL
LIN {X 0,Y 367.253,Z 525.307,A -85,B 0,C 180,E1 -12556.652,E2 -12556.652} C_VEL
LIN {X 0,Y 367.271,Z 525.328,A -85,B 0,C 180,E1 -12558.271,E2 -12558.271} C_VEL
LIN {X 0,Y 367.34,Z 524.418,A -85,B 0,C 180,E1 -12559.933,E2 -12559.933} C_VEL
LIN {X 0,Y 367.608,Z 522.533,A -85,B 0,C 180,E1 -12561.615,E2 -12561.615} C_VEL
LIN {X 0,Y 368.01,Z 518.789,A -85,B 0,C 180,E1 -12563.699,E2 -12563.699} C_VEL
LIN {X 0,Y 368.426,Z 515.321,A -85,B 0,C 180,E1 -12565.111,E2 -12565.111} C_VEL
LIN {X 0,Y 369.054,Z 509.567,A -85,B 0,C 180,E1 -12566.92,E2 -12566.92} C_VEL
LIN {X 0,Y 369.911,Z 502.069,A -85,B 0,C 180,E1 -12568.756,E2 -12568.756} C_VEL
LIN {X 0,Y 370.783,Z 494.901,A -85,B 0,C 180,E1 -12570.161,E2 -12570.161} C_VEL
LIN {X 0,Y 371.803,Z 485.614,A -85,B 0,C 180,E1 -12571.645,E2 -12571.645} C_VEL
LIN {X 0,Y 372.836,Z 475.127,A -85,B 0,C 180,E1 -12572.996,E2 -12572.996} C_VEL
LIN {X 0,Y 373.939,Z 464.17,A -85,B 0,C 180,E1 -12574.119,E2 -12574.119} C_VEL
LIN {X 0,Y 374.888,Z 452.536,A -85,B 0,C 180,E1 -12575.051,E2 -12575.051} C_VEL
LIN {X 0,Y 375.682,Z 440.574,A -85,B 0,C 180,E1 -12575.781,E2 -12575.781} C_VEL
LIN {X 0,Y 376.23,Z 427.66,A -85,B 0,C 180,E1 -12576.349,E2 -12576.349} C_VEL
LIN {X 0,Y 376.713,Z 412.739,A -85,B 0,C 180,E1 -12576.734,E2 -12576.734} C_VEL
LIN {X 0,Y 378.453,Z 338.965,A -85,B 0,C 180,E1 -12578.295,E2 -12578.295} C_VEL
LIN {X 0,Y 375.183,Z 323.938,A -85,B 0,C 180,E1 -12578.88,E2 -12578.88} C_VEL
LIN {X 0,Y 371.313,Z 314.295,A -85,B 0,C 180,E1 -12579.43,E2 -12579.43} C_VEL
LIN {X 0,Y 368.99,Z 304.527,A -85,B 0,C 180,E1 -12581.841,E2 -12581.841} C_VEL
LIN {X 0,Y 369.018,Z 304.524,A -85,B 0,C 180,E1 -12585.665,E2 -12585.665} C_VEL
LIN {X 0,Y 369.023,Z 304.519,A -85,B 0,C 180,E1 -12589.021,E2 -12589.021} C_VEL
LIN {X 0,Y 369.19,Z 304.498,A -85,B 0,C 180,E1 -12592.342,E2 -12592.342} C_VEL
LIN {X 0,Y 369.145,Z 304.503,A -85,B 0,C 180,E1 -12594.537,E2 -12594.537} C_VEL
LIN {X 0,Y 369.318,Z 304.481,A -85,B 0,C 180,E1 -12597.819,E2 -12597.819} C_VEL
LIN {X 0,Y 369.458,Z 304.464,A -85,B 0,C 180,E1 -12600,E2 -12600} C_VEL
LIN {X 0,Y 369.318,Z 304.484,A -85,B 0,C 180,E1 -12602.181,E2 -12602.181} C_VEL
LIN {X 0,Y 369.18,Z 304.492,A -85,B 0,C 180,E1 -12606.558,E2 -12606.558} C_VEL
LIN {X 0,Y 369.069,Z 304.509,A -85,B 0,C 180,E1 -12609.868,E2 -12609.868} C_VEL
LIN {X 0,Y 369.039,Z 304.509,A -85,B 0,C 180,E1 -12613.772,E2 -12613.772} C_VEL
LIN {X 0,Y 368.992,Z 304.514,A -85,B 0,C 180,E1 -12617.743,E2 -12617.743} C_VEL
LIN {X 0,Y 368.912,Z 304.526,A -85,B 0,C 180,E1 -12621.221,E2 -12621.221} C_VEL
LIN {X 0,Y 368.957,Z 304.52,A -85,B 0,C 180,E1 -12624.775,E2 -12624.775} C_VEL
LIN {X 0,Y 368.965,Z 304.519,A -85,B 0,C 180,E1 -12627.203,E2 -12627.203} C_VEL
LIN {X 0,Y 368.931,Z 304.525,A -85,B 0,C 180,E1 -12630.953,E2 -12630.953} C_VEL
LIN {X 0,Y 368.93,Z 304.526,A -85,B 0,C 180,E1 -12635.001,E2 -12635.001} C_VEL
LIN {X 0,Y 368.909,Z 304.529,A -85,B 0,C 180,E1 -12638.64,E2 -12638.64} C_VEL
LIN {X 0,Y 368.883,Z 304.535,A -85,B 0,C 180,E1 -12642.009,E2 -12642.009} C_VEL
LIN {X 0,Y 368.882,Z 304.538,A -85,B 0,C 180,E1 -12645.176,E2 -12645.176} C_VEL
LIN {X 0,Y 368.884,Z 304.533,A -85,B 0,C 180,E1 -12648.177,E2 -12648.177} C_VEL
LIN {X 0,Y 368.909,Z 304.535,A -85,B 0,C 180,E1 -12651.36,E2 -12651.36} C_VEL
LIN {X 0,Y 368.939,Z 304.533,A -85,B 0,C 180,E1 -12655.146,E2 -12655.146} C_VEL
LIN {X 0,Y 368.931,Z 304.533,A -85,B 0,C 180,E1 -12659.046,E2 -12659.046} C_VEL
LIN {X 0,Y 368.943,Z 304.665,A -85,B 0,C 180,E1 -12659.879,E2 -12659.879} C_VEL
LIN {X 0,Y 371.311,Z 314.461,A -85,B 0,C 180,E1 -12662.334,E2 -12662.334} C_VEL
LIN {X 0,Y 372.931,Z 322.75,A -85,B 0,C 180,E1 -12664.313,E2 -12664.313} C_VEL
LIN {X 0,Y 372.983,Z 326.347,A -85,B 0,C 180,E1 -12665.108,E2 -12665.108} C_VEL
LIN {X 0,Y 371.925,Z 338.543,A -85,B 0,C 180,E1 -12667.692,E2 -12667.692} C_VEL
LIN {X 0,Y 375.888,Z 359.93,A -85,B 0,C 180,E1 -12668.489,E2 -12668.489} C_VEL
LIN {X 0,Y 377.818,Z 373.266,A -85,B 0,C 180,E1 -12668.927,E2 -12668.927} C_VEL
LIN {X 0,Y 376.116,Z 448.933,A -85,B 0,C 180,E1 -12670.558,E2 -12670.558} C_VEL
LIN {X 0,Y 375.31,Z 462.913,A -85,B 0,C 180,E1 -12671.083,E2 -12671.083} C_VEL
LIN {X 0,Y 374.363,Z 475.877,A -85,B 0,C 180,E1 -12671.813,E2 -12671.813} C_VEL
LIN {X 0,Y 373.25,Z 488.185,A -85,B 0,C 180,E1 -12672.748,E2 -12672.748} C_VEL
LIN {X 0,Y 372.139,Z 499.276,A -85,B 0,C 180,E1 -12673.825,E2 -12673.825} C_VEL
LIN {X 0,Y 371.049,Z 509.923,A -85,B 0,C 180,E1 -12675.132,E2 -12675.132} C_VEL
LIN {X 0,Y 370.086,Z 519.267,A -85,B 0,C 180,E1 -12676.548,E2 -12676.548} C_VEL
LIN {X 0,Y 369.034,Z 528.04,A -85,B 0,C 180,E1 -12678.186,E2 -12678.186} C_VEL
LIN {X 0,Y 368.329,Z 535.062,A -85,B 0,C 180,E1 -12679.834,E2 -12679.834} C_VEL
LIN {X 0,Y 367.84,Z 541.535,A -85,B 0,C 180,E1 -12681.761,E2 -12681.761} C_VEL
LIN {X 0,Y 367.563,Z 545.782,A -85,B 0,C 180,E1 -12683.412,E2 -12683.412} C_VEL
LIN {X 0,Y 367.465,Z 548.024,A -85,B 0,C 180,E1 -12684.512,E2 -12684.512} C_VEL
LIN {X 0,Y 367.456,Z 549.787,A -85,B 0,C 180,E1 -12685.612,E2 -12685.612} C_VEL
LIN {X 0,Y 367.396,Z 552.086,A -85,B 0,C 180,E1 -12687.807,E2 -12687.807} C_VEL
LIN {X 0,Y 367.468,Z 552.599,A -85,B 0,C 180,E1 -12688.903,E2 -12688.903} C_VEL
LIN {X 0,Y 367.506,Z 552.69,A -85,B 0,C 180,E1 -12689.999,E2 -12689.999} C_VEL
LIN {X 0,Y 367.484,Z 552.381,A -85,B 0,C 180,E1 -12691.095,E2 -12691.095} C_VEL
LIN {X 0,Y 367.402,Z 551.67,A -85,B 0,C 180,E1 -12692.192,E2 -12692.192} C_VEL
LIN {X 0,Y 367.385,Z 550.509,A -85,B 0,C 180,E1 -12693.289,E2 -12693.289} C_VEL
LIN {X 0,Y 367.463,Z 547.975,A -85,B 0,C 180,E1 -12694.937,E2 -12694.937} C_VEL
LIN {X 0,Y 367.563,Z 544.392,A -85,B 0,C 180,E1 -12696.587,E2 -12696.587} C_VEL
LIN {X 0,Y 367.795,Z 539.666,A -85,B 0,C 180,E1 -12698.239,E2 -12698.239} C_VEL
LIN {X 0,Y 368.193,Z 533.658,A -85,B 0,C 180,E1 -12699.891,E2 -12699.891} C_VEL
LIN {X 0,Y 368.783,Z 526.151,A -85,B 0,C 180,E1 -12701.542,E2 -12701.542} C_VEL
LIN {X 0,Y 369.519,Z 518.499,A -85,B 0,C 180,E1 -12702.913,E2 -12702.913} C_VEL
LIN {X 0,Y 370.344,Z 509.218,A -85,B 0,C 180,E1 -12704.282,E2 -12704.282} C_VEL
LIN {X 0,Y 371.165,Z 498.879,A -85,B 0,C 180,E1 -12705.512,E2 -12705.512} C_VEL
LIN {X 0,Y 372.107,Z 487.437,A -85,B 0,C 180,E1 -12706.598,E2 -12706.598} C_VEL
LIN {X 0,Y 373.019,Z 475.581,A -85,B 0,C 180,E1 -12707.473,E2 -12707.473} C_VEL
LIN {X 0,Y 373.824,Z 462.566,A -85,B 0,C 180,E1 -12708.177,E2 -12708.177} C_VEL
LIN {X 0,Y 374.473,Z 448.852,A -85,B 0,C 180,E1 -12708.676,E2 -12708.676} C_VEL
LIN {X 0,Y 375.767,Z 372.598,A -85,B 0,C 180,E1 -12710.273,E2 -12710.273} C_VEL
LIN {X 0,Y 371.101,Z 340.59,A -85,B 0,C 180,E1 -12711.206,E2 -12711.206} C_VEL
LIN {X 0,Y 372.441,Z 325.581,A -85,B 0,C 180,E1 -12714.527,E2 -12714.527} C_VEL
LIN {X 0,Y 372.48,Z 321.977,A -85,B 0,C 180,E1 -12715.348,E2 -12715.348} C_VEL
LIN {X 0,Y 370.064,Z 309.718,A -85,B 0,C 180,E1 -12718.344,E2 -12718.344} C_VEL
LIN {X 0,Y 368.94,Z 304.531,A -85,B 0,C 180,E1 -12719.687,E2 -12719.687} C_VEL
LIN {X 0,Y 368.896,Z 304.531,A -85,B 0,C 180,E1 -12723.537,E2 -12723.537} C_VEL
LIN {X 0,Y 368.898,Z 304.531,A -85,B 0,C 180,E1 -12726.855,E2 -12726.855} C_VEL
LIN {X 0,Y 368.907,Z 304.535,A -85,B 0,C 180,E1 -12730.369,E2 -12730.369} C_VEL
LIN {X 0,Y 368.879,Z 304.532,A -85,B 0,C 180,E1 -12733.615,E2 -12733.615} C_VEL
LIN {X 0,Y 368.883,Z 304.536,A -85,B 0,C 180,E1 -12736.695,E2 -12736.695} C_VEL
LIN {X 0,Y 368.909,Z 304.528,A -85,B 0,C 180,E1 -12739.642,E2 -12739.642} C_VEL
LIN {X 0,Y 368.898,Z 304.532,A -85,B 0,C 180,E1 -12743.143,E2 -12743.143} C_VEL
LIN {X 0,Y 368.891,Z 304.533,A -85,B 0,C 180,E1 -12746.461,E2 -12746.461} C_VEL
LIN {X 0,Y 368.924,Z 304.531,A -85,B 0,C 180,E1 -12749.046,E2 -12749.046} C_VEL
LIN {X 0,Y 368.957,Z 304.527,A -85,B 0,C 180,E1 -12752.796,E2 -12752.796} C_VEL
LIN {X 0,Y 368.94,Z 304.524,A -85,B 0,C 180,E1 -12756.113,E2 -12756.113} C_VEL
LIN {X 0,Y 368.93,Z 304.526,A -85,B 0,C 180,E1 -12759.947,E2 -12759.947} C_VEL
LIN {X 0,Y 368.971,Z 304.526,A -85,B 0,C 180,E1 -12763.399,E2 -12763.399} C_VEL
LIN {X 0,Y 369.052,Z 304.511,A -85,B 0,C 180,E1 -12766.79,E2 -12766.79} C_VEL
LIN {X 0,Y 369.062,Z 304.51,A -85,B 0,C 180,E1 -12770.132,E2 -12770.132} C_VEL
LIN {X 0,Y 369.182,Z 304.494,A -85,B 0,C 180,E1 -12772.342,E2 -12772.342} C_VEL
LIN {X 0,Y 369.138,Z 304.499,A -85,B 0,C 180,E1 -12774.538,E2 -12774.538} C_VEL
LIN {X 0,Y 369.31,Z 304.483,A -85,B 0,C 180,E1 -12777.819,E2 -12777.819} C_VEL
LIN {X 0,Y 369.45,Z 304.464,A -85,B 0,C 180,E1 -12780,E2 -12780} C_VEL
LIN {X 0,Y 369.311,Z 304.48,A -85,B 0,C 180,E1 -12782.181,E2 -12782.181} C_VEL
LIN {X 0,Y 369.172,Z 304.496,A -85,B 0,C 180,E1 -12786.559,E2 -12786.559} C_VEL
LIN {X 0,Y 369.062,Z 304.515,A -85,B 0,C 180,E1 -12789.869,E2 -12789.869} C_VEL
LIN {X 0,Y 369.032,Z 304.516,A -85,B 0,C 180,E1 -12793.773,E2 -12793.773} C_VEL
LIN {X 0,Y 368.996,Z 304.519,A -85,B 0,C 180,E1 -12797.769,E2 -12797.769} C_VEL
LIN {X 0,Y 368.905,Z 304.528,A -85,B 0,C 180,E1 -12801.222,E2 -12801.222} C_VEL
LIN {X 0,Y 368.928,Z 304.528,A -85,B 0,C 180,E1 -12804.778,E2 -12804.778} C_VEL
LIN {X 0,Y 368.912,Z 304.534,A -85,B 0,C 180,E1 -12808.442,E2 -12808.442} C_VEL
LIN {X 0,Y 368.907,Z 304.531,A -85,B 0,C 180,E1 -12810.988,E2 -12810.988} C_VEL
LIN {X 0,Y 368.933,Z 304.53,A -85,B 0,C 180,E1 -12814.854,E2 -12814.854} C_VEL
LIN {X 0,Y 368.879,Z 304.537,A -85,B 0,C 180,E1 -12818.636,E2 -12818.636} C_VEL
LIN {X 0,Y 368.877,Z 304.532,A -85,B 0,C 180,E1 -12822.01,E2 -12822.01} C_VEL
LIN {X 0,Y 368.877,Z 304.536,A -85,B 0,C 180,E1 -12825.177,E2 -12825.177} C_VEL
LIN {X 0,Y 368.868,Z 304.533,A -85,B 0,C 180,E1 -12828.177,E2 -12828.177} C_VEL
LIN {X 0,Y 368.877,Z 304.536,A -85,B 0,C 180,E1 -12831.367,E2 -12831.367} C_VEL
LIN {X 0,Y 368.936,Z 304.531,A -85,B 0,C 180,E1 -12835.148,E2 -12835.148} C_VEL
LIN {X 0,Y 368.913,Z 304.531,A -85,B 0,C 180,E1 -12839.046,E2 -12839.046} C_VEL
LIN {X 0,Y 368.908,Z 304.533,A -85,B 0,C 180,E1 -12841.559,E2 -12841.559} C_VEL
LIN {X 0,Y 368.915,Z 304.531,A -85,B 0,C 180,E1 -12845.222,E2 -12845.222} C_VEL
LIN {X 0,Y 368.912,Z 304.528,A -85,B 0,C 180,E1 -12848.78,E2 -12848.78} C_VEL
LIN {X 0,Y 368.993,Z 304.519,A -85,B 0,C 180,E1 -12852.258,E2 -12852.258} C_VEL
LIN {X 0,Y 369.04,Z 304.514,A -85,B 0,C 180,E1 -12856.229,E2 -12856.229} C_VEL
LIN {X 0,Y 369.061,Z 304.513,A -85,B 0,C 180,E1 -12860.132,E2 -12860.132} C_VEL
